LIN {X 0,Y 532.462,Z 881.05,A -85,B 0,C 180,E1 15618.4,E2 15618.4} C_VEL
LIN {X 0,Y 529.556,Z 900.929,A -85,B 0,C 180,E1 15617.745,E2 15617.745} C_VEL
LIN {X 0,Y 525.913,Z 922.421,A -85,B 0,C 180,E1 15616.892,E2 15616.892} C_VEL
LIN {X 0,Y 520.896,Z 948,A -85,B 0,C 180,E1 15615.653,E2 15615.653} C_VEL
LIN {X 0,Y 516.441,Z 968.016,A -85,B 0,C 180,E1 15614.497,E2 15614.497} C_VEL
LIN {X 0,Y 511.868,Z 987.021,A -85,B 0,C 180,E1 15613.228,E2 15613.228} C_VEL
LIN {X 0,Y 506.208,Z 1009.005,A -85,B 0,C 180,E1 15611.528,E2 15611.528} C_VEL
LIN {X 0,Y 500.786,Z 1028.462,A -85,B 0,C 180,E1 15609.762,E2 15609.762} C_VEL
LIN {X 0,Y 495.987,Z 1045.107,A -85,B 0,C 180,E1 15608.041,E2 15608.041} C_VEL
LIN {X 0,Y 490.456,Z 1064.014,A -85,B 0,C 180,E1 15605.81,E2 15605.81} C_VEL
LIN {X 0,Y 489.126,Z 1068.218,A -85,B 0,C 180,E1 15605.252,E2 15605.252} C_VEL
LIN {X 0,Y 486.734,Z 1073.439,A -85,B 0,C 180,E1 15604.629,E2 15604.629} C_VEL
LIN {X 0,Y 477.301,Z 1087.199,A -85,B 0,C 180,E1 15603.072,E2 15603.072} C_VEL
LIN {X 0,Y 475.397,Z 1091.188,A -85,B 0,C 180,E1 15602.478,E2 15602.478} C_VEL
LIN {X 0,Y 471.344,Z 1104.372,A -85,B 0,C 180,E1 15600.183,E2 15600.183} C_VEL
LIN {X 0,Y 467.671,Z 1116.791,A -85,B 0,C 180,E1 15597.731,E2 15597.731} C_VEL
LIN {X 0,Y 463.729,Z 1130.988,A -85,B 0,C 180,E1 15594.456,E2 15594.456} C_VEL
LIN {X 0,Y 461.345,Z 1140.474,A -85,B 0,C 180,E1 15591.887,E2 15591.887} C_VEL
LIN {X 0,Y 459.415,Z 1149.184,A -85,B 0,C 180,E1 15589.164,E2 15589.164} C_VEL
LIN {X 0,Y 457.712,Z 1158.339,A -85,B 0,C 180,E1 15585.717,E2 15585.717} C_VEL
LIN {X 0,Y 456.832,Z 1164.35,A -85,B 0,C 180,E1 15582.9,E2 15582.9} C_VEL
LIN {X 0,Y 456.324,Z 1168.956,A -85,B 0,C 180,E1 15580.223,E2 15580.223} C_VEL
LIN {X 0,Y 456.055,Z 1172.944,A -85,B 0,C 180,E1 15577.179,E2 15577.179} C_VEL
LIN {X 0,Y 455.949,Z 1175.579,A -85,B 0,C 180,E1 15573.898,E2 15573.898} C_VEL
LIN {X 0,Y 455.936,Z 1176.585,A -85,B 0,C 180,E1 15571.257,E2 15571.257} C_VEL
LIN {X 0,Y 455.939,Z 1176.6,A -85,B 0,C 180,E1 15568.744,E2 15568.744} C_VEL
LIN {X 0,Y 455.942,Z 1175.69,A -85,B 0,C 180,E1 15566.225,E2 15566.225} C_VEL
LIN {X 0,Y 456.031,Z 1173.527,A -85,B 0,C 180,E1 15563.327,E2 15563.327} C_VEL
LIN {X 0,Y 456.288,Z 1169.494,A -85,B 0,C 180,E1 15560.031,E2 15560.031} C_VEL
LIN {X 0,Y 456.784,Z 1164.768,A -85,B 0,C 180,E1 15557.228,E2 15557.228} C_VEL
LIN {X 0,Y 457.573,Z 1159.13,A -85,B 0,C 180,E1 15554.539,E2 15554.539} C_VEL
LIN {X 0,Y 459.07,Z 1150.955,A -85,B 0,C 180,E1 15551.327,E2 15551.327} C_VEL
LIN {X 0,Y 461.171,Z 1141.22,A -85,B 0,C 180,E1 15548.238,E2 15548.238} C_VEL
LIN {X 0,Y 463.506,Z 1131.822,A -85,B 0,C 180,E1 15545.668,E2 15545.668} C_VEL
LIN {X 0,Y 467.018,Z 1119.253,A -85,B 0,C 180,E1 15542.688,E2 15542.688} C_VEL
LIN {X 0,Y 471.007,Z 1105.511,A -85,B 0,C 180,E1 15539.935,E2 15539.935} C_VEL
LIN {X 0,Y 474.943,Z 1092.667,A -85,B 0,C 180,E1 15537.674,E2 15537.674} C_VEL
LIN {X 0,Y 480.115,Z 1076.281,A -85,B 0,C 180,E1 15535.14,E2 15535.14} C_VEL
LIN {X 0,Y 485.422,Z 1059.029,A -85,B 0,C 180,E1 15532.86,E2 15532.86} C_VEL
LIN {X 0,Y 490.456,Z 1042.604,A -85,B 0,C 180,E1 15530.954,E2 15530.954} C_VEL
LIN {X 0,Y 496.369,Z 1022.898,A -85,B 0,C 180,E1 15528.953,E2 15528.953} C_VEL
LIN {X 0,Y 502.173,Z 1002.09,A -85,B 0,C 180,E1 15527.16,E2 15527.16} C_VEL
LIN {X 0,Y 506.959,Z 983.945,A -85,B 0,C 180,E1 15525.797,E2 15525.797} C_VEL
LIN {X 0,Y 512.003,Z 963.456,A -85,B 0,C 180,E1 15524.457,E2 15524.457} C_VEL
LIN {X 0,Y 517.286,Z 939.51,A -85,B 0,C 180,E1 15523.141,E2 15523.141} C_VEL
LIN {X 0,Y 521.291,Z 918.889,A -85,B 0,C 180,E1 15522.188,E2 15522.188} C_VEL
LIN {X 0,Y 524.924,Z 897.699,A -85,B 0,C 180,E1 15521.367,E2 15521.367} C_VEL
LIN {X 0,Y 528.667,Z 871.635,A -85,B 0,C 180,E1 15520.555,E2 15520.555} C_VEL
LIN {X 0,Y 531.302,Z 847.596,A -85,B 0,C 180,E1 15519.993,E2 15519.993} C_VEL
LIN {X 0,Y 533.012,Z 825.454,A -85,B 0,C 180,E1 15519.597,E2 15519.597} C_VEL
LIN {X 0,Y 543.801,Z 591.304,A -85,B 0,C 180,E1 15516.126,E2 15516.126} C_VEL
LIN {X 0,Y 549.38,Z 477.095,A -85,B 0,C 180,E1 15514.411,E2 15514.411} C_VEL
LIN {X 0,Y 538.923,Z 460.101,A -85,B 0,C 180,E1 15512.174,E2 15512.174} C_VEL
LIN {X 0,Y 528.718,Z 444.717,A -85,B 0,C 180,E1 15509.77,E2 15509.77} C_VEL
LIN {X 0,Y 520.734,Z 433.186,A -85,B 0,C 180,E1 15507.69,E2 15507.69} C_VEL
LIN {X 0,Y 514.214,Z 424.156,A -85,B 0,C 180,E1 15505.822,E2 15505.822} C_VEL
LIN {X 0,Y 509.213,Z 417.399,A -85,B 0,C 180,E1 15504.26,E2 15504.26} C_VEL
LIN {X 0,Y 503.323,Z 409.516,A -85,B 0,C 180,E1 15502.231,E2 15502.231} C_VEL
LIN {X 0,Y 498.472,Z 403.274,A -85,B 0,C 180,E1 15500.367,E2 15500.367} C_VEL
LIN {X 0,Y 494.802,Z 398.678,A -85,B 0,C 180,E1 15498.803,E2 15498.803} C_VEL
LIN {X 0,Y 490.932,Z 393.536,A -85,B 0,C 180,E1 15496.933,E2 15496.933} C_VEL
LIN {X 0,Y 487.374,Z 389.283,A -85,B 0,C 180,E1 15494.981,E2 15494.981} C_VEL
LIN {X 0,Y 485.876,Z 387.485,A -85,B 0,C 180,E1 15494.054,E2 15494.054} C_VEL
LIN {X 0,Y 481.885,Z 382.272,A -85,B 0,C 180,E1 15491.057,E2 15491.057} C_VEL
LIN {X 0,Y 477.66,Z 376.715,A -85,B 0,C 180,E1 15485.646,E2 15485.646} C_VEL
LIN {X 0,Y 476.978,Z 375.814,A -85,B 0,C 180,E1 15481.081,E2 15481.081} C_VEL
LIN {X 0,Y 478.968,Z 376.994,A -85,B 0,C 180,E1 15476.649,E2 15476.649} C_VEL
LIN {X 0,Y 480.364,Z 378.25,A -85,B 0,C 180,E1 15474.985,E2 15474.985} C_VEL
LIN {X 0,Y 486.543,Z 384.476,A -85,B 0,C 180,E1 15470.119,E2 15470.119} C_VEL
LIN {X 0,Y 490.446,Z 388.953,A -85,B 0,C 180,E1 15467.878,E2 15467.878} C_VEL
LIN {X 0,Y 492.385,Z 390.817,A -85,B 0,C 180,E1 15466.913,E2 15466.913} C_VEL
LIN {X 0,Y 495.897,Z 395.017,A -85,B 0,C 180,E1 15465.282,E2 15465.282} C_VEL
LIN {X 0,Y 497.624,Z 396.68,A -85,B 0,C 180,E1 15464.559,E2 15464.559} C_VEL
LIN {X 0,Y 501.643,Z 401.372,A -85,B 0,C 180,E1 15462.962,E2 15462.962} C_VEL
LIN {X 0,Y 508.034,Z 409.049,A -85,B 0,C 180,E1 15460.692,E2 15460.692} C_VEL
LIN {X 0,Y 512.753,Z 414.817,A -85,B 0,C 180,E1 15459.182,E2 15459.182} C_VEL
LIN {X 0,Y 517.573,Z 420.901,A -85,B 0,C 180,E1 15457.75,E2 15457.75} C_VEL
LIN {X 0,Y 524.781,Z 430.02,A -85,B 0,C 180,E1 15455.787,E2 15455.787} C_VEL
LIN {X 0,Y 534.925,Z 443.868,A -85,B 0,C 180,E1 15453.285,E2 15453.285} C_VEL
LIN {X 0,Y 544.949,Z 458.293,A -85,B 0,C 180,E1 15451.057,E2 15451.057} C_VEL
LIN {X 0,Y 552.935,Z 470.605,A -85,B 0,C 180,E1 15449.413,E2 15449.413} C_VEL
LIN {X 0,Y 541.839,Z 683.901,A -85,B 0,C 180,E1 15446.095,E2 15446.095} C_VEL
LIN {X 0,Y 534.574,Z 826.583,A -85,B 0,C 180,E1 15443.866,E2 15443.866} C_VEL
LIN {X 0,Y 532.122,Z 853.861,A -85,B 0,C 180,E1 15443.33,E2 15443.33} C_VEL
LIN {X 0,Y 528.759,Z 880.247,A -85,B 0,C 180,E1 15442.619,E2 15442.619} C_VEL
LIN {X 0,Y 525.469,Z 902.039,A -85,B 0,C 180,E1 15441.889,E2 15441.889} C_VEL
LIN {X 0,Y 521.778,Z 923.361,A -85,B 0,C 180,E1 15441.035,E2 15441.035} C_VEL
LIN {X 0,Y 516.644,Z 949.664,A -85,B 0,C 180,E1 15439.772,E2 15439.772} C_VEL
LIN {X 0,Y 511.586,Z 972.397,A -85,B 0,C 180,E1 15438.465,E2 15438.465} C_VEL
LIN {X 0,Y 506.827,Z 992.36,A -85,B 0,C 180,E1 15437.143,E2 15437.143} C_VEL
LIN {X 0,Y 501.686,Z 1012.679,A -85,B 0,C 180,E1 15435.608,E2 15435.608} C_VEL
LIN {X 0,Y 495.251,Z 1036.643,A -85,B 0,C 180,E1 15433.507,E2 15433.507} C_VEL
LIN {X 0,Y 490.026,Z 1055.322,A -85,B 0,C 180,E1 15431.618,E2 15431.618} C_VEL
LIN {X 0,Y 485.244,Z 1072.171,A -85,B 0,C 180,E1 15429.7,E2 15429.7} C_VEL
LIN {X 0,Y 479.749,Z 1091.705,A -85,B 0,C 180,E1 15427.186,E2 15427.186} C_VEL
LIN {X 0,Y 474.635,Z 1109.565,A -85,B 0,C 180,E1 15424.519,E2 15424.519} C_VEL
LIN {X 0,Y 470.851,Z 1123.31,A -85,B 0,C 180,E1 15422.209,E2 15422.209} C_VEL
LIN {X 0,Y 467.156,Z 1137.727,A -85,B 0,C 180,E1 15419.49,E2 15419.49} C_VEL
LIN {X 0,Y 463.668,Z 1152.034,A -85,B 0,C 180,E1 15416.374,E2 15416.374} C_VEL
LIN {X 0,Y 461.39,Z 1162.388,A -85,B 0,C 180,E1 15413.771,E2 15413.771} C_VEL
LIN {X 0,Y 459.598,Z 1171.455,A -85,B 0,C 180,E1 15411.17,E2 15411.17} C_VEL
LIN {X 0,Y 458.241,Z 1179.295,A -85,B 0,C 180,E1 15408.576,E2 15408.576} C_VEL
LIN {X 0,Y 457.218,Z 1186.471,A -85,B 0,C 180,E1 15405.795,E2 15405.795} C_VEL
LIN {X 0,Y 456.438,Z 1193.644,A -85,B 0,C 180,E1 15402.396,E2 15402.396} C_VEL
LIN {X 0,Y 456.093,Z 1198.482,A -85,B 0,C 180,E1 15399.336,E2 15399.336} C_VEL
LIN {X 0,Y 455.961,Z 1201.688,A -85,B 0,C 180,E1 15396.585,E2 15396.585} C_VEL
LIN {X 0,Y 455.915,Z 1203.684,A -85,B 0,C 180,E1 15394.024,E2 15394.024} C_VEL
LIN {X 0,Y 455.91,Z 1204.708,A -85,B 0,C 180,E1 15391.508,E2 15391.508} C_VEL
LIN {X 0,Y 455.908,Z 1204.801,A -85,B 0,C 180,E1 15388.994,E2 15388.994} C_VEL
LIN {X 0,Y 455.915,Z 1203.964,A -85,B 0,C 180,E1 15386.479,E2 15386.479} C_VEL
LIN {X 0,Y 455.946,Z 1202.191,A -85,B 0,C 180,E1 15383.957,E2 15383.957} C_VEL
LIN {X 0,Y 456.045,Z 1199.471,A -85,B 0,C 180,E1 15381.426,E2 15381.426} C_VEL
LIN {X 0,Y 456.253,Z 1195.782,A -85,B 0,C 180,E1 15378.88,E2 15378.88} C_VEL
LIN {X 0,Y 456.713,Z 1190.833,A -85,B 0,C 180,E1 15376.194,E2 15376.194} C_VEL
LIN {X 0,Y 457.385,Z 1185.054,A -85,B 0,C 180,E1 15373.62,E2 15373.62} C_VEL
LIN {X 0,Y 458.489,Z 1177.83,A -85,B 0,C 180,E1 15370.906,E2 15370.906} C_VEL
LIN {X 0,Y 460.348,Z 1167.648,A -85,B 0,C 180,E1 15367.66,E2 15367.66} C_VEL
LIN {X 0,Y 462.817,Z 1155.82,A -85,B 0,C 180,E1 15364.537,E2 15364.537} C_VEL
LIN {X 0,Y 465.352,Z 1144.907,A -85,B 0,C 180,E1 15362.02,E2 15362.02} C_VEL
LIN {X 0,Y 468.293,Z 1133.073,A -85,B 0,C 180,E1 15359.6,E2 15359.6} C_VEL
LIN {X 0,Y 472.647,Z 1117.012,A -85,B 0,C 180,E1 15356.682,E2 15356.682} C_VEL
LIN {X 0,Y 477.455,Z 1099.47,A -85,B 0,C 180,E1 15353.937,E2 15353.937} C_VEL
LIN {X 0,Y 481.832,Z 1084.082,A -85,B 0,C 180,E1 15351.801,E2 15351.801} C_VEL
LIN {X 0,Y 486.748,Z 1066.938,A -85,B 0,C 180,E1 15349.679,E2 15349.679} C_VEL
LIN {X 0,Y 493.233,Z 1043.981,A -85,B 0,C 180,E1 15347.211,E2 15347.211} C_VEL
LIN {X 0,Y 498.131,Z 1026.031,A -85,B 0,C 180,E1 15345.53,E2 15345.53} C_VEL
LIN {X 0,Y 502.839,Z 1008.166,A -85,B 0,C 180,E1 15344.042,E2 15344.042} C_VEL
LIN {X 0,Y 507.623,Z 989.113,A -85,B 0,C 180,E1 15342.634,E2 15342.634} C_VEL
LIN {X 0,Y 513.346,Z 964.927,A -85,B 0,C 180,E1 15341.08,E2 15341.08} C_VEL
LIN {X 0,Y 518.424,Z 940.627,A -85,B 0,C 180,E1 15339.773,E2 15339.773} C_VEL
LIN {X 0,Y 522.355,Z 919.986,A -85,B 0,C 180,E1 15338.824,E2 15338.824} C_VEL
LIN {X 0,Y 525.919,Z 899.053,A -85,B 0,C 180,E1 15338.005,E2 15338.005} C_VEL
LIN {X 0,Y 529.858,Z 872.442,A -85,B 0,C 180,E1 15337.15,E2 15337.15} C_VEL
LIN {X 0,Y 532.806,Z 846.446,A -85,B 0,C 180,E1 15336.517,E2 15336.517} C_VEL
LIN {X 0,Y 534.717,Z 823.813,A -85,B 0,C 180,E1 15336.091,E2 15336.091} C_VEL
LIN {X 0,Y 545.542,Z 610.54,A -85,B 0,C 180,E1 15332.769,E2 15332.769} C_VEL
LIN {X 0,Y 552.772,Z 470.258,A -85,B 0,C 180,E1 15330.567,E2 15330.567} C_VEL
LIN {X 0,Y 542.221,Z 454.418,A -85,B 0,C 180,E1 15328.38,E2 15328.38} C_VEL
LIN {X 0,Y 532.873,Z 440.999,A -85,B 0,C 180,E1 15326.255,E2 15326.255} C_VEL
LIN {X 0,Y 523.322,Z 428.23,A -85,B 0,C 180,E1 15323.865,E2 15323.865} C_VEL
LIN {X 0,Y 515.323,Z 417.986,A -85,B 0,C 180,E1 15321.633,E2 15321.633} C_VEL
LIN {X 0,Y 510.35,Z 411.91,A -85,B 0,C 180,E1 15320.111,E2 15320.111} C_VEL
LIN {X 0,Y 506.154,Z 406.806,A -85,B 0,C 180,E1 15318.724,E2 15318.724} C_VEL
LIN {X 0,Y 501.489,Z 401.24,A -85,B 0,C 180,E1 15317.043,E2 15317.043} C_VEL
LIN {X 0,Y 497.404,Z 396.37,A -85,B 0,C 180,E1 15315.418,E2 15315.418} C_VEL
LIN {X 0,Y 492.888,Z 391.636,A -85,B 0,C 180,E1 15313.431,E2 15313.431} C_VEL
LIN {X 0,Y 491.406,Z 389.729,A -85,B 0,C 180,E1 15312.695,E2 15312.695} C_VEL
LIN {X 0,Y 486.891,Z 385.029,A -85,B 0,C 180,E1 15310.232,E2 15310.232} C_VEL
LIN {X 0,Y 485.71,Z 383.571,A -85,B 0,C 180,E1 15309.479,E2 15309.479} C_VEL
LIN {X 0,Y 479.508,Z 377.269,A -85,B 0,C 180,E1 15304.305,E2 15304.305} C_VEL
LIN {X 0,Y 476.828,Z 375.617,A -85,B 0,C 180,E1 15299.519,E2 15299.519} C_VEL
LIN {X 0,Y 477.071,Z 376.199,A -85,B 0,C 180,E1 15295.07,E2 15295.07} C_VEL
LIN {X 0,Y 477.957,Z 377.33,A -85,B 0,C 180,E1 15293.151,E2 15293.151} C_VEL
LIN {X 0,Y 482.557,Z 383.147,A -85,B 0,C 180,E1 15288.102,E2 15288.102} C_VEL
LIN {X 0,Y 487.234,Z 389.112,A -85,B 0,C 180,E1 15284.893,E2 15284.893} C_VEL
LIN {X 0,Y 490.92,Z 393.558,A -85,B 0,C 180,E1 15282.884,E2 15282.884} C_VEL
LIN {X 0,Y 496.633,Z 401.015,A -85,B 0,C 180,E1 15280.23,E2 15280.23} C_VEL
LIN {X 0,Y 500.623,Z 406.102,A -85,B 0,C 180,E1 15278.623,E2 15278.623} C_VEL
LIN {X 0,Y 505.172,Z 411.999,A -85,B 0,C 180,E1 15276.961,E2 15276.961} C_VEL
LIN {X 0,Y 512.277,Z 421.55,A -85,B 0,C 180,E1 15274.632,E2 15274.632} C_VEL
LIN {X 0,Y 518.676,Z 430.345,A -85,B 0,C 180,E1 15272.752,E2 15272.752} C_VEL
LIN {X 0,Y 527.608,Z 443.059,A -85,B 0,C 180,E1 15270.386,E2 15270.386} C_VEL
LIN {X 0,Y 538.197,Z 459.107,A -85,B 0,C 180,E1 15267.872,E2 15267.872} C_VEL
LIN {X 0,Y 548.067,Z 474.977,A -85,B 0,C 180,E1 15265.748,E2 15265.748} C_VEL
LIN {X 0,Y 549.35,Z 477.405,A -85,B 0,C 180,E1 15265.478,E2 15265.478} C_VEL
LIN {X 0,Y 538.35,Z 706.811,A -85,B 0,C 180,E1 15262.067,E2 15262.067} C_VEL
LIN {X 0,Y 532.598,Z 831.176,A -85,B 0,C 180,E1 15260.216,E2 15260.216} C_VEL
LIN {X 0,Y 530.219,Z 858.217,A -85,B 0,C 180,E1 15259.683,E2 15259.683} C_VEL
LIN {X 0,Y 527.373,Z 880.936,A -85,B 0,C 180,E1 15259.078,E2 15259.078} C_VEL
LIN {X 0,Y 524.411,Z 900.63,A -85,B 0,C 180,E1 15258.43,E2 15258.43} C_VEL
LIN {X 0,Y 520.708,Z 921.873,A -85,B 0,C 180,E1 15257.589,E2 15257.589} C_VEL
LIN {X 0,Y 515.429,Z 948.057,A -85,B 0,C 180,E1 15256.321,E2 15256.321} C_VEL
LIN {X 0,Y 510.955,Z 967.573,A -85,B 0,C 180,E1 15255.192,E2 15255.192} C_VEL
LIN {X 0,Y 506.155,Z 986.915,A -85,B 0,C 180,E1 15253.898,E2 15253.898} C_VEL
LIN {X 0,Y 500.279,Z 1008.979,A -85,B 0,C 180,E1 15252.187,E2 15252.187} C_VEL
LIN {X 0,Y 494.655,Z 1028.456,A -85,B 0,C 180,E1 15250.408,E2 15250.408} C_VEL
LIN {X 0,Y 489.663,Z 1045.152,A -85,B 0,C 180,E1 15248.671,E2 15248.671} C_VEL
LIN {X 0,Y 483.962,Z 1063.92,A -85,B 0,C 180,E1 15246.44,E2 15246.44} C_VEL
LIN {X 0,Y 478.537,Z 1081.053,A -85,B 0,C 180,E1 15244.054,E2 15244.054} C_VEL
LIN {X 0,Y 475.397,Z 1091.188,A -85,B 0,C 180,E1 15242.478,E2 15242.478} C_VEL
LIN {X 0,Y 473.094,Z 1095.843,A -85,B 0,C 180,E1 15241.776,E2 15241.776} C_VEL
LIN {X 0,Y 463.841,Z 1108.186,A -85,B 0,C 180,E1 15239.993,E2 15239.993} C_VEL
LIN {X 0,Y 462.049,Z 1111.733,A -85,B 0,C 180,E1 15239.332,E2 15239.332} C_VEL
LIN {X 0,Y 458.366,Z 1123.819,A -85,B 0,C 180,E1 15236.703,E2 15236.703} C_VEL
LIN {X 0,Y 455.419,Z 1134.273,A -85,B 0,C 180,E1 15234.102,E2 15234.102} C_VEL
LIN {X 0,Y 452.577,Z 1145.51,A -85,B 0,C 180,E1 15230.836,E2 15230.836} C_VEL
LIN {X 0,Y 450.692,Z 1154.074,A -85,B 0,C 180,E1 15227.828,E2 15227.828} C_VEL
LIN {X 0,Y 449.497,Z 1160.654,A -85,B 0,C 180,E1 15225.086,E2 15225.086} C_VEL
LIN {X 0,Y 448.613,Z 1167.046,A -85,B 0,C 180,E1 15221.833,E2 15221.833} C_VEL
LIN {X 0,Y 448.177,Z 1171.674,A -85,B 0,C 180,E1 15218.597,E2 15218.597} C_VEL
LIN {X 0,Y 447.993,Z 1174.46,A -85,B 0,C 180,E1 15215.893,E2 15215.893} C_VEL
LIN {X 0,Y 447.945,Z 1176.219,A -85,B 0,C 180,E1 15213.199,E2 15213.199} C_VEL
LIN {X 0,Y 447.936,Z 1177.029,A -85,B 0,C 180,E1 15210.128,E2 15210.128} C_VEL
LIN {X 0,Y 447.943,Z 1176.331,A -85,B 0,C 180,E1 15206.929,E2 15206.929} C_VEL
LIN {X 0,Y 447.993,Z 1174.539,A -85,B 0,C 180,E1 15204.107,E2 15204.107} C_VEL
LIN {X 0,Y 448.169,Z 1171.783,A -85,B 0,C 180,E1 15201.404,E2 15201.404} C_VEL
LIN {X 0,Y 448.547,Z 1167.582,A -85,B 0,C 180,E1 15198.427,E2 15198.427} C_VEL
LIN {X 0,Y 449.424,Z 1161.15,A -85,B 0,C 180,E1 15195.044,E2 15195.044} C_VEL
LIN {X 0,Y 450.582,Z 1154.652,A -85,B 0,C 180,E1 15192.301,E2 15192.301} C_VEL
LIN {X 0,Y 452.224,Z 1146.949,A -85,B 0,C 180,E1 15189.553,E2 15189.553} C_VEL
LIN {X 0,Y 454.955,Z 1136.099,A -85,B 0,C 180,E1 15186.285,E2 15186.285} C_VEL
LIN {X 0,Y 458.093,Z 1124.745,A -85,B 0,C 180,E1 15183.42,E2 15183.42} C_VEL
LIN {X 0,Y 461.456,Z 1113.604,A -85,B 0,C 180,E1 15180.964,E2 15180.964} C_VEL
LIN {X 0,Y 466.102,Z 1098.989,A -85,B 0,C 180,E1 15178.149,E2 15178.149} C_VEL
LIN {X 0,Y 471.039,Z 1083.585,A -85,B 0,C 180,E1 15175.623,E2 15175.623} C_VEL
LIN {X 0,Y 475.822,Z 1068.929,A -85,B 0,C 180,E1 15173.51,E2 15173.51} C_VEL
LIN {X 0,Y 481.805,Z 1050.577,A -85,B 0,C 180,E1 15171.191,E2 15171.191} C_VEL
LIN {X 0,Y 487.874,Z 1030.932,A -85,B 0,C 180,E1 15169.081,E2 15169.081} C_VEL
LIN {X 0,Y 492.905,Z 1014.172,A -85,B 0,C 180,E1 15167.507,E2 15167.507} C_VEL
LIN {X 0,Y 498.692,Z 993.945,A -85,B 0,C 180,E1 15165.843,E2 15165.843} C_VEL
LIN {X 0,Y 504.647,Z 970.976,A -85,B 0,C 180,E1 15164.246,E2 15164.246} C_VEL
LIN {X 0,Y 509.316,Z 951.469,A -85,B 0,C 180,E1 15163.089,E2 15163.089} C_VEL
LIN {X 0,Y 513.751,Z 931.077,A -85,B 0,C 180,E1 15162.048,E2 15162.048} C_VEL
LIN {X 0,Y 518.582,Z 905.394,A -85,B 0,C 180,E1 15160.963,E2 15160.963} C_VEL
LIN {X 0,Y 521.939,Z 884.167,A -85,B 0,C 180,E1 15160.238,E2 15160.238} C_VEL
LIN {X 0,Y 524.617,Z 863.87,A -85,B 0,C 180,E1 15159.672,E2 15159.672} C_VEL
LIN {X 0,Y 527.172,Z 839.566,A -85,B 0,C 180,E1 15159.145,E2 15159.145} C_VEL
LIN {X 0,Y 529.271,Z 803.306,A -85,B 0,C 180,E1 15158.57,E2 15158.57} C_VEL
LIN {X 0,Y 540.117,Z 575.69,A -85,B 0,C 180,E1 15155.184,E2 15155.184} C_VEL
LIN {X 0,Y 544.866,Z 481.213,A -85,B 0,C 180,E1 15153.751,E2 15153.751} C_VEL
LIN {X 0,Y 535.364,Z 465.745,A -85,B 0,C 180,E1 15151.656,E2 15151.656} C_VEL
LIN {X 0,Y 525.934,Z 451.284,A -85,B 0,C 180,E1 15149.374,E2 15149.374} C_VEL
LIN {X 0,Y 518.091,Z 439.848,A -85,B 0,C 180,E1 15147.282,E2 15147.282} C_VEL
LIN {X 0,Y 512.035,Z 431.315,A -85,B 0,C 180,E1 15145.505,E2 15145.505} C_VEL
LIN {X 0,Y 505.61,Z 422.408,A -85,B 0,C 180,E1 15143.422,E2 15143.422} C_VEL
LIN {X 0,Y 501.184,Z 416.583,A -85,B 0,C 180,E1 15141.844,E2 15141.844} C_VEL
LIN {X 0,Y 496.7,Z 410.664,A -85,B 0,C 180,E1 15140.074,E2 15140.074} C_VEL
LIN {X 0,Y 493.095,Z 406.104,A -85,B 0,C 180,E1 15138.503,E2 15138.503} C_VEL
LIN {X 0,Y 489.413,Z 401.142,A -85,B 0,C 180,E1 15136.681,E2 15136.681} C_VEL
LIN {X 0,Y 485.846,Z 396.679,A -85,B 0,C 180,E1 15134.663,E2 15134.663} C_VEL
LIN {X 0,Y 480.729,Z 390.107,A -85,B 0,C 180,E1 15130.911,E2 15130.911} C_VEL
LIN {X 0,Y 476.638,Z 384.614,A -85,B 0,C 180,E1 15125.538,E2 15125.538} C_VEL
LIN {X 0,Y 476.019,Z 383.758,A -85,B 0,C 180,E1 15120.963,E2 15120.963} C_VEL
LIN {X 0,Y 478.172,Z 385.043,A -85,B 0,C 180,E1 15116.403,E2 15116.403} C_VEL
LIN {X 0,Y 479.485,Z 386.415,A -85,B 0,C 180,E1 15114.855,E2 15114.855} C_VEL
LIN {X 0,Y 485.192,Z 392.155,A -85,B 0,C 180,E1 15110.331,E2 15110.331} C_VEL
LIN {X 0,Y 489.244,Z 396.837,A -85,B 0,C 180,E1 15107.968,E2 15107.968} C_VEL
LIN {X 0,Y 490.93,Z 398.526,A -85,B 0,C 180,E1 15107.113,E2 15107.113} C_VEL
LIN {X 0,Y 494.526,Z 402.811,A -85,B 0,C 180,E1 15105.42,E2 15105.42} C_VEL
LIN {X 0,Y 496.223,Z 404.609,A -85,B 0,C 180,E1 15104.694,E2 15104.694} C_VEL
LIN {X 0,Y 501.221,Z 410.498,A -85,B 0,C 180,E1 15102.708,E2 15102.708} C_VEL
LIN {X 0,Y 506.311,Z 416.724,A -85,B 0,C 180,E1 15100.893,E2 15100.893} C_VEL
LIN {X 0,Y 510.814,Z 422.288,A -85,B 0,C 180,E1 15099.429,E2 15099.429} C_VEL
LIN {X 0,Y 515.576,Z 428.38,A -85,B 0,C 180,E1 15097.989,E2 15097.989} C_VEL
LIN {X 0,Y 522.515,Z 437.285,A -85,B 0,C 180,E1 15096.066,E2 15096.066} C_VEL
LIN {X 0,Y 532.238,Z 450.725,A -85,B 0,C 180,E1 15093.621,E2 15093.621} C_VEL
LIN {X 0,Y 542.138,Z 465.167,A -85,B 0,C 180,E1 15091.375,E2 15091.375} C_VEL
LIN {X 0,Y 548.391,Z 474.999,A -85,B 0,C 180,E1 15090.051,E2 15090.051} C_VEL
LIN {X 0,Y 536.927,Z 688.4,A -85,B 0,C 180,E1 15086.718,E2 15086.718} C_VEL
LIN {X 0,Y 529.646,Z 826.679,A -85,B 0,C 180,E1 15084.547,E2 15084.547} C_VEL
LIN {X 0,Y 527.109,Z 854.091,A -85,B 0,C 180,E1 15084.007,E2 15084.007} C_VEL
LIN {X 0,Y 523.677,Z 880.287,A -85,B 0,C 180,E1 15083.299,E2 15083.299} C_VEL
LIN {X 0,Y 520.312,Z 901.929,A -85,B 0,C 180,E1 15082.573,E2 15082.573} C_VEL
LIN {X 0,Y 516.536,Z 923.116,A -85,B 0,C 180,E1 15081.724,E2 15081.724} C_VEL
LIN {X 0,Y 511.332,Z 949.047,A -85,B 0,C 180,E1 15080.481,E2 15080.481} C_VEL
LIN {X 0,Y 505.911,Z 972.651,A -85,B 0,C 180,E1 15079.118,E2 15079.118} C_VEL
LIN {X 0,Y 501.16,Z 991.953,A -85,B 0,C 180,E1 15077.832,E2 15077.832} C_VEL
LIN {X 0,Y 496.053,Z 1011.473,A -85,B 0,C 180,E1 15076.354,E2 15076.354} C_VEL
LIN {X 0,Y 489.551,Z 1034.938,A -85,B 0,C 180,E1 15074.307,E2 15074.307} C_VEL
LIN {X 0,Y 483.912,Z 1054.308,A -85,B 0,C 180,E1 15072.345,E2 15072.345} C_VEL
LIN {X 0,Y 478.907,Z 1071.214,A -85,B 0,C 180,E1 15070.411,E2 15070.411} C_VEL
LIN {X 0,Y 473.735,Z 1088.691,A -85,B 0,C 180,E1 15068.159,E2 15068.159} C_VEL
LIN {X 0,Y 468.048,Z 1107.914,A -85,B 0,C 180,E1 15065.307,E2 15065.307} C_VEL
LIN {X 0,Y 463.915,Z 1122.151,A -85,B 0,C 180,E1 15062.897,E2 15062.897} C_VEL
LIN {X 0,Y 460.461,Z 1134.589,A -85,B 0,C 180,E1 15060.539,E2 15060.539} C_VEL
LIN {X 0,Y 456.978,Z 1148.192,A -85,B 0,C 180,E1 15057.636,E2 15057.636} C_VEL
LIN {X 0,Y 453.828,Z 1161.463,A -85,B 0,C 180,E1 15054.33,E2 15054.33} C_VEL
LIN {X 0,Y 451.904,Z 1170.658,A -85,B 0,C 180,E1 15051.673,E2 15051.673} C_VEL
LIN {X 0,Y 450.46,Z 1178.567,A -85,B 0,C 180,E1 15049.044,E2 15049.044} C_VEL
LIN {X 0,Y 449.393,Z 1185.361,A -85,B 0,C 180,E1 15046.413,E2 15046.413} C_VEL
LIN {X 0,Y 448.68,Z 1191.316,A -85,B 0,C 180,E1 15043.663,E2 15043.663} C_VEL
LIN {X 0,Y 448.187,Z 1196.991,A -85,B 0,C 180,E1 15040.411,E2 15040.411} C_VEL
LIN {X 0,Y 447.974,Z 1201.111,A -85,B 0,C 180,E1 15037.051,E2 15037.051} C_VEL
LIN {X 0,Y 447.92,Z 1203.361,A -85,B 0,C 180,E1 15034.224,E2 15034.224} C_VEL
LIN {X 0,Y 447.911,Z 1204.436,A -85,B 0,C 180,E1 15031.663,E2 15031.663} C_VEL
LIN {X 0,Y 447.908,Z 1204.577,A -85,B 0,C 180,E1 15029.104,E2 15029.104} C_VEL
LIN {X 0,Y 447.917,Z 1203.714,A -85,B 0,C 180,E1 15026.416,E2 15026.416} C_VEL
LIN {X 0,Y 447.951,Z 1201.935,A -85,B 0,C 180,E1 15023.849,E2 15023.849} C_VEL
LIN {X 0,Y 448.054,Z 1199.204,A -85,B 0,C 180,E1 15021.271,E2 15021.271} C_VEL
LIN {X 0,Y 448.275,Z 1195.5,A -85,B 0,C 180,E1 15018.68,E2 15018.68} C_VEL
LIN {X 0,Y 448.736,Z 1190.793,A -85,B 0,C 180,E1 15016.075,E2 15016.075} C_VEL
LIN {X 0,Y 449.436,Z 1185.044,A -85,B 0,C 180,E1 15013.455,E2 15013.455} C_VEL
LIN {X 0,Y 450.589,Z 1177.838,A -85,B 0,C 180,E1 15010.692,E2 15010.692} C_VEL
LIN {X 0,Y 452.466,Z 1167.953,A -85,B 0,C 180,E1 15007.478,E2 15007.478} C_VEL
LIN {X 0,Y 455.107,Z 1155.88,A -85,B 0,C 180,E1 15004.214,E2 15004.214} C_VEL
LIN {X 0,Y 457.835,Z 1144.603,A -85,B 0,C 180,E1 15001.569,E2 15001.569} C_VEL
LIN {X 0,Y 461.011,Z 1132.611,A -85,B 0,C 180,E1 14999.067,E2 14999.067} C_VEL
LIN {X 0,Y 465.426,Z 1117.066,A -85,B 0,C 180,E1 14996.192,E2 14996.192} C_VEL
LIN {X 0,Y 470.343,Z 1099.999,A -85,B 0,C 180,E1 14993.47,E2 14993.47} C_VEL
LIN {X 0,Y 474.917,Z 1084.606,A -85,B 0,C 180,E1 14991.296,E2 14991.296} C_VEL
LIN {X 0,Y 479.692,Z 1068.587,A -85,B 0,C 180,E1 14989.275,E2 14989.275} C_VEL
LIN {X 0,Y 485.84,Z 1047.993,A -85,B 0,C 180,E1 14986.981,E2 14986.981} C_VEL
LIN {X 0,Y 491.792,Z 1026.909,A -85,B 0,C 180,E1 14984.965,E2 14984.965} C_VEL
LIN {X 0,Y 496.619,Z 1009.281,A -85,B 0,C 180,E1 14983.477,E2 14983.477} C_VEL
LIN {X 0,Y 501.369,Z 991.052,A -85,B 0,C 180,E1 14982.108,E2 14982.108} C_VEL
LIN {X 0,Y 506.393,Z 970.579,A -85,B 0,C 180,E1 14980.756,E2 14980.756} C_VEL
LIN {X 0,Y 512.247,Z 944.525,A -85,B 0,C 180,E1 14979.29,E2 14979.29} C_VEL
LIN {X 0,Y 516.742,Z 921.818,A -85,B 0,C 180,E1 14978.224,E2 14978.224} C_VEL
LIN {X 0,Y 520.426,Z 901.019,A -85,B 0,C 180,E1 14977.397,E2 14977.397} C_VEL
LIN {X 0,Y 523.856,Z 878.838,A -85,B 0,C 180,E1 14976.66,E2 14976.66} C_VEL
LIN {X 0,Y 527.386,Z 850.986,A -85,B 0,C 180,E1 14975.93,E2 14975.93} C_VEL
LIN {X 0,Y 529.658,Z 825.826,A -85,B 0,C 180,E1 14975.442,E2 14975.442} C_VEL
LIN {X 0,Y 540.247,Z 624.464,A -85,B 0,C 180,E1 14972.288,E2 14972.288} C_VEL
LIN {X 0,Y 548.34,Z 474.693,A -85,B 0,C 180,E1 14969.949,E2 14969.949} C_VEL
LIN {X 0,Y 536.551,Z 456.942,A -85,B 0,C 180,E1 14967.406,E2 14967.406} C_VEL
LIN {X 0,Y 527.28,Z 443.875,A -85,B 0,C 180,E1 14965.197,E2 14965.197} C_VEL
LIN {X 0,Y 518.102,Z 431.461,A -85,B 0,C 180,E1 14962.765,E2 14962.765} C_VEL
LIN {X 0,Y 509.027,Z 419.974,A -85,B 0,C 180,E1 14960.046,E2 14960.046} C_VEL
LIN {X 0,Y 504.065,Z 414.015,A -85,B 0,C 180,E1 14958.385,E2 14958.385} C_VEL
LIN {X 0,Y 499.625,Z 408.646,A -85,B 0,C 180,E1 14956.749,E2 14956.749} C_VEL
LIN {X 0,Y 494.884,Z 403.11,A -85,B 0,C 180,E1 14954.808,E2 14954.808} C_VEL
LIN {X 0,Y 491.086,Z 398.824,A -85,B 0,C 180,E1 14953.062,E2 14953.062} C_VEL
LIN {X 0,Y 489.964,Z 397.43,A -85,B 0,C 180,E1 14952.493,E2 14952.493} C_VEL
LIN {X 0,Y 485.526,Z 392.707,A -85,B 0,C 180,E1 14950.022,E2 14950.022} C_VEL
LIN {X 0,Y 484.363,Z 391.323,A -85,B 0,C 180,E1 14949.266,E2 14949.266} C_VEL
LIN {X 0,Y 478.422,Z 385.155,A -85,B 0,C 180,E1 14944.195,E2 14944.195} C_VEL
LIN {X 0,Y 475.821,Z 383.549,A -85,B 0,C 180,E1 14939.398,E2 14939.398} C_VEL
LIN {X 0,Y 476.141,Z 384.191,A -85,B 0,C 180,E1 14934.94,E2 14934.94} C_VEL
LIN {X 0,Y 476.979,Z 385.348,A -85,B 0,C 180,E1 14933.137,E2 14933.137} C_VEL
LIN {X 0,Y 481.374,Z 390.961,A -85,B 0,C 180,E1 14928.255,E2 14928.255} C_VEL
LIN {X 0,Y 485.883,Z 396.823,A -85,B 0,C 180,E1 14925.094,E2 14925.094} C_VEL
LIN {X 0,Y 489.628,Z 401.368,A -85,B 0,C 180,E1 14923.021,E2 14923.021} C_VEL
LIN {X 0,Y 495.405,Z 409.108,A -85,B 0,C 180,E1 14920.302,E2 14920.302} C_VEL
LIN {X 0,Y 498.948,Z 413.692,A -85,B 0,C 180,E1 14918.855,E2 14918.855} C_VEL
LIN {X 0,Y 503.37,Z 419.507,A -85,B 0,C 180,E1 14917.21,E2 14917.21} C_VEL
LIN {X 0,Y 510.206,Z 428.834,A -85,B 0,C 180,E1 14914.925,E2 14914.925} C_VEL
LIN {X 0,Y 516.431,Z 437.517,A -85,B 0,C 180,E1 14913.06,E2 14913.06} C_VEL
LIN {X 0,Y 525.324,Z 450.408,A -85,B 0,C 180,E1 14910.658,E2 14910.658} C_VEL
LIN {X 0,Y 535.611,Z 466.172,A -85,B 0,C 180,E1 14908.171,E2 14908.171} C_VEL
LIN {X 0,Y 544.889,Z 481.344,A -85,B 0,C 180,E1 14906.132,E2 14906.132} C_VEL
LIN {X 0,Y 533.478,Z 711.175,A -85,B 0,C 180,E1 14902.701,E2 14902.701} C_VEL
LIN {X 0,Y 527.72,Z 831.166,A -85,B 0,C 180,E1 14900.904,E2 14900.904} C_VEL
LIN {X 0,Y 525.272,Z 858.21,A -85,B 0,C 180,E1 14900.371,E2 14900.371} C_VEL
LIN {X 0,Y 522.344,Z 880.922,A -85,B 0,C 180,E1 14899.766,E2 14899.766} C_VEL
LIN {X 0,Y 519.196,Z 901.222,A -85,B 0,C 180,E1 14899.096,E2 14899.096} C_VEL
LIN {X 0,Y 515.354,Z 922.588,A -85,B 0,C 180,E1 14898.245,E2 14898.245} C_VEL
LIN {X 0,Y 509.999,Z 948.263,A -85,B 0,C 180,E1 14896.994,E2 14896.994} C_VEL
LIN {X 0,Y 505.224,Z 968.436,A -85,B 0,C 180,E1 14895.819,E2 14895.819} C_VEL
LIN {X 0,Y 500.246,Z 987.835,A -85,B 0,C 180,E1 14894.51,E2 14894.51} C_VEL
LIN {X 0,Y 493.712,Z 1011.303,A -85,B 0,C 180,E1 14892.652,E2 14892.652} C_VEL
LIN {X 0,Y 488.217,Z 1029.68,A -85,B 0,C 180,E1 14890.948,E2 14890.948} C_VEL
LIN {X 0,Y 482.862,Z 1046.951,A -85,B 0,C 180,E1 14889.12,E2 14889.12} C_VEL
LIN {X 0,Y 476.608,Z 1066.534,A -85,B 0,C 180,E1 14886.72,E2 14886.72} C_VEL
LIN {X 0,Y 471.738,Z 1081.397,A -85,B 0,C 180,E1 14884.614,E2 14884.614} C_VEL
LIN {X 0,Y 467.164,Z 1095.495,A -85,B 0,C 180,E1 14882.349,E2 14882.349} C_VEL
LIN {X 0,Y 462.375,Z 1110.731,A -85,B 0,C 180,E1 14879.541,E2 14879.541} C_VEL
LIN {X 0,Y 462.049,Z 1111.733,A -85,B 0,C 180,E1 14879.332,E2 14879.332} C_VEL
LIN {X 0,Y 459.887,Z 1115.797,A -85,B 0,C 180,E1 14878.553,E2 14878.553} C_VEL
LIN {X 0,Y 450.982,Z 1126.66,A -85,B 0,C 180,E1 14876.548,E2 14876.548} C_VEL
LIN {X 0,Y 449.349,Z 1129.716,A -85,B 0,C 180,E1 14875.824,E2 14875.824} C_VEL
LIN {X 0,Y 446.217,Z 1140.62,A -85,B 0,C 180,E1 14872.809,E2 14872.809} C_VEL
LIN {X 0,Y 444.029,Z 1149.305,A -85,B 0,C 180,E1 14870.016,E2 14870.016} C_VEL
LIN {X 0,Y 442.119,Z 1158.309,A -85,B 0,C 180,E1 14866.556,E2 14866.556} C_VEL
LIN {X 0,Y 441.01,Z 1164.787,A -85,B 0,C 180,E1 14863.427,E2 14863.427} C_VEL
LIN {X 0,Y 440.408,Z 1169.483,A -85,B 0,C 180,E1 14860.597,E2 14860.597} C_VEL
LIN {X 0,Y 440.097,Z 1173.459,A -85,B 0,C 180,E1 14857.441,E2 14857.441} C_VEL
LIN {X 0,Y 439.961,Z 1176.078,A -85,B 0,C 180,E1 14854.04,E2 14854.04} C_VEL
LIN {X 0,Y 439.942,Z 1177.079,A -85,B 0,C 180,E1 14851.303,E2 14851.303} C_VEL
LIN {X 0,Y 439.946,Z 1177.095,A -85,B 0,C 180,E1 14848.698,E2 14848.698} C_VEL
LIN {X 0,Y 439.954,Z 1176.19,A -85,B 0,C 180,E1 14846.091,E2 14846.091} C_VEL
LIN {X 0,Y 440.048,Z 1174.131,A -85,B 0,C 180,E1 14843.203,E2 14843.203} C_VEL
LIN {X 0,Y 440.342,Z 1170.215,A -85,B 0,C 180,E1 14839.799,E2 14839.799} C_VEL
LIN {X 0,Y 440.938,Z 1165.302,A -85,B 0,C 180,E1 14836.76,E2 14836.76} C_VEL
LIN {X 0,Y 441.855,Z 1159.676,A -85,B 0,C 180,E1 14833.974,E2 14833.974} C_VEL
LIN {X 0,Y 443.552,Z 1151.522,A -85,B 0,C 180,E1 14830.648,E2 14830.648} C_VEL
LIN {X 0,Y 445.906,Z 1141.802,A -85,B 0,C 180,E1 14827.453,E2 14827.453} C_VEL
LIN {X 0,Y 448.512,Z 1132.415,A -85,B 0,C 180,E1 14824.799,E2 14824.799} C_VEL
LIN {X 0,Y 452.325,Z 1120.05,A -85,B 0,C 180,E1 14821.768,E2 14821.768} C_VEL
LIN {X 0,Y 456.888,Z 1105.835,A -85,B 0,C 180,E1 14818.837,E2 14818.837} C_VEL
LIN {X 0,Y 461.334,Z 1092.569,A -85,B 0,C 180,E1 14816.45,E2 14816.45} C_VEL
LIN {X 0,Y 467.128,Z 1075.596,A -85,B 0,C 180,E1 14813.789,E2 14813.789} C_VEL
LIN {X 0,Y 472.952,Z 1058.207,A -85,B 0,C 180,E1 14811.466,E2 14811.466} C_VEL
LIN {X 0,Y 478.217,Z 1042.265,A -85,B 0,C 180,E1 14809.597,E2 14809.597} C_VEL
LIN {X 0,Y 484.785,Z 1021.789,A -85,B 0,C 180,E1 14807.509,E2 14807.509} C_VEL
LIN {X 0,Y 490.609,Z 1002.247,A -85,B 0,C 180,E1 14805.813,E2 14805.813} C_VEL
LIN {X 0,Y 495.498,Z 984.886,A -85,B 0,C 180,E1 14804.493,E2 14804.493} C_VEL
LIN {X 0,Y 500.621,Z 965.359,A -85,B 0,C 180,E1 14803.197,E2 14803.197} C_VEL
LIN {X 0,Y 506.703,Z 939.626,A -85,B 0,C 180,E1 14801.763,E2 14801.763} C_VEL
LIN {X 0,Y 511.049,Z 918.479,A -85,B 0,C 180,E1 14800.785,E2 14800.785} C_VEL
LIN {X 0,Y 514.897,Z 897.154,A -85,B 0,C 180,E1 14799.958,E2 14799.958} C_VEL
LIN {X 0,Y 519.039,Z 869.339,A -85,B 0,C 180,E1 14799.107,E2 14799.107} C_VEL
LIN {X 0,Y 521.638,Z 846.653,A -85,B 0,C 180,E1 14798.584,E2 14798.584} C_VEL
LIN {X 0,Y 523.468,Z 823.805,A -85,B 0,C 180,E1 14798.178,E2 14798.178} C_VEL
LIN {X 0,Y 535.074,Z 589.3,A -85,B 0,C 180,E1 14794.67,E2 14794.67} C_VEL
LIN {X 0,Y 540.486,Z 485.434,A -85,B 0,C 180,E1 14793.093,E2 14793.093} C_VEL
LIN {X 0,Y 529.694,Z 467.828,A -85,B 0,C 180,E1 14790.611,E2 14790.611} C_VEL
LIN {X 0,Y 519.738,Z 452.688,A -85,B 0,C 180,E1 14788.059,E2 14788.059} C_VEL
LIN {X 0,Y 510.737,Z 439.567,A -85,B 0,C 180,E1 14785.45,E2 14785.45} C_VEL
LIN {X 0,Y 503.55,Z 429.596,A -85,B 0,C 180,E1 14783.09,E2 14783.09} C_VEL
LIN {X 0,Y 499.348,Z 423.967,A -85,B 0,C 180,E1 14781.558,E2 14781.558} C_VEL
LIN {X 0,Y 494.939,Z 418.059,A -85,B 0,C 180,E1 14779.779,E2 14779.779} C_VEL
LIN {X 0,Y 491.402,Z 413.525,A -85,B 0,C 180,E1 14778.2,E2 14778.2} C_VEL
LIN {X 0,Y 488.061,Z 408.89,A -85,B 0,C 180,E1 14776.509,E2 14776.509} C_VEL
LIN {X 0,Y 484.507,Z 404.392,A -85,B 0,C 180,E1 14774.46,E2 14774.46} C_VEL
LIN {X 0,Y 479.631,Z 397.991,A -85,B 0,C 180,E1 14770.814,E2 14770.814} C_VEL
LIN {X 0,Y 475.619,Z 392.515,A -85,B 0,C 180,E1 14765.429,E2 14765.429} C_VEL
LIN {X 0,Y 475.063,Z 391.702,A -85,B 0,C 180,E1 14760.844,E2 14760.844} C_VEL
LIN {X 0,Y 477.288,Z 393.05,A -85,B 0,C 180,E1 14756.276,E2 14756.276} C_VEL
LIN {X 0,Y 478.828,Z 394.928,A -85,B 0,C 180,E1 14754.488,E2 14754.488} C_VEL
LIN {X 0,Y 483.934,Z 399.972,A -85,B 0,C 180,E1 14750.486,E2 14750.486} C_VEL
LIN {X 0,Y 488.044,Z 404.72,A -85,B 0,C 180,E1 14748.058,E2 14748.058} C_VEL
LIN {X 0,Y 489.484,Z 406.232,A -85,B 0,C 180,E1 14747.315,E2 14747.315} C_VEL
LIN {X 0,Y 493.288,Z 410.717,A -85,B 0,C 180,E1 14745.503,E2 14745.503} C_VEL
LIN {X 0,Y 494.827,Z 412.52,A -85,B 0,C 180,E1 14744.83,E2 14744.83} C_VEL
LIN {X 0,Y 499.566,Z 418.149,A -85,B 0,C 180,E1 14742.919,E2 14742.919} C_VEL
LIN {X 0,Y 504.442,Z 424.177,A -85,B 0,C 180,E1 14741.15,E2 14741.15} C_VEL
LIN {X 0,Y 508.968,Z 429.869,A -85,B 0,C 180,E1 14739.652,E2 14739.652} C_VEL
LIN {X 0,Y 513.765,Z 436.089,A -85,B 0,C 180,E1 14738.178,E2 14738.178} C_VEL
LIN {X 0,Y 520.638,Z 445.086,A -85,B 0,C 180,E1 14736.245,E2 14736.245} C_VEL
LIN {X 0,Y 529.668,Z 457.735,A -85,B 0,C 180,E1 14733.936,E2 14733.936} C_VEL
LIN {X 0,Y 539.345,Z 472.039,A -85,B 0,C 180,E1 14731.697,E2 14731.697} C_VEL
LIN {X 0,Y 543.914,Z 479.375,A -85,B 0,C 180,E1 14730.7,E2 14730.7} C_VEL
LIN {X 0,Y 532.127,Z 692.058,A -85,B 0,C 180,E1 14727.366,E2 14727.366} C_VEL
LIN {X 0,Y 524.802,Z 826.684,A -85,B 0,C 180,E1 14725.243,E2 14725.243} C_VEL
LIN {X 0,Y 522.202,Z 854.102,A -85,B 0,C 180,E1 14724.701,E2 14724.701} C_VEL
LIN {X 0,Y 518.693,Z 880.192,A -85,B 0,C 180,E1 14723.997,E2 14723.997} C_VEL
LIN {X 0,Y 515.232,Z 901.833,A -85,B 0,C 180,E1 14723.271,E2 14723.271} C_VEL
LIN {X 0,Y 511.447,Z 922.51,A -85,B 0,C 180,E1 14722.443,E2 14722.443} C_VEL
LIN {X 0,Y 506.252,Z 947.838,A -85,B 0,C 180,E1 14721.237,E2 14721.237} C_VEL
LIN {X 0,Y 500.567,Z 971.876,A -85,B 0,C 180,E1 14719.851,E2 14719.851} C_VEL
LIN {X 0,Y 495.607,Z 991.43,A -85,B 0,C 180,E1 14718.546,E2 14718.546} C_VEL
LIN {X 0,Y 490.735,Z 1009.478,A -85,B 0,C 180,E1 14717.181,E2 14717.181} C_VEL
LIN {X 0,Y 485.229,Z 1028.858,A -85,B 0,C 180,E1 14715.523,E2 14715.523} C_VEL
LIN {X 0,Y 478.26,Z 1052.157,A -85,B 0,C 180,E1 14713.213,E2 14713.213} C_VEL
LIN {X 0,Y 472.995,Z 1069.234,A -85,B 0,C 180,E1 14711.265,E2 14711.265} C_VEL
LIN {X 0,Y 468.042,Z 1085.167,A -85,B 0,C 180,E1 14709.223,E2 14709.223} C_VEL
LIN {X 0,Y 462.644,Z 1102.669,A -85,B 0,C 180,E1 14706.695,E2 14706.695} C_VEL
LIN {X 0,Y 457.279,Z 1120.31,A -85,B 0,C 180,E1 14703.737,E2 14703.737} C_VEL
LIN {X 0,Y 453.387,Z 1133.531,A -85,B 0,C 180,E1 14701.215,E2 14701.215} C_VEL
LIN {X 0,Y 450.08,Z 1145.46,A -85,B 0,C 180,E1 14698.654,E2 14698.654} C_VEL
LIN {X 0,Y 446.782,Z 1158.621,A -85,B 0,C 180,E1 14695.447,E2 14695.447} C_VEL
LIN {X 0,Y 444.236,Z 1169.795,A -85,B 0,C 180,E1 14692.218,E2 14692.218} C_VEL
LIN {X 0,Y 442.689,Z 1177.823,A -85,B 0,C 180,E1 14689.528,E2 14689.528} C_VEL
LIN {X 0,Y 441.542,Z 1184.699,A -85,B 0,C 180,E1 14686.849,E2 14686.849} C_VEL
LIN {X 0,Y 440.823,Z 1190.218,A -85,B 0,C 180,E1 14684.314,E2 14684.314} C_VEL
LIN {X 0,Y 440.322,Z 1195.001,A -85,B 0,C 180,E1 14681.659,E2 14681.659} C_VEL
LIN {X 0,Y 440.072,Z 1198.768,A -85,B 0,C 180,E1 14679.019,E2 14679.019} C_VEL
LIN {X 0,Y 439.959,Z 1201.558,A -85,B 0,C 180,E1 14676.393,E2 14676.393} C_VEL
LIN {X 0,Y 439.92,Z 1203.391,A -85,B 0,C 180,E1 14673.779,E2 14673.779} C_VEL
LIN {X 0,Y 439.919,Z 1204.283,A -85,B 0,C 180,E1 14671.172,E2 14671.172} C_VEL
LIN {X 0,Y 439.921,Z 1204.26,A -85,B 0,C 180,E1 14668.697,E2 14668.697} C_VEL
LIN {X 0,Y 439.92,Z 1203.322,A -85,B 0,C 180,E1 14666.09,E2 14666.09} C_VEL
LIN {X 0,Y 439.963,Z 1201.441,A -85,B 0,C 180,E1 14663.475,E2 14663.475} C_VEL
LIN {X 0,Y 440.079,Z 1198.603,A -85,B 0,C 180,E1 14660.848,E2 14660.848} C_VEL
LIN {X 0,Y 440.343,Z 1194.786,A -85,B 0,C 180,E1 14658.208,E2 14658.208} C_VEL
LIN {X 0,Y 440.886,Z 1189.695,A -85,B 0,C 180,E1 14655.42,E2 14655.42} C_VEL
LIN {X 0,Y 441.864,Z 1182.708,A -85,B 0,C 180,E1 14652.304,E2 14652.304} C_VEL
LIN {X 0,Y 443.65,Z 1172.77,A -85,B 0,C 180,E1 14648.724,E2 14648.724} C_VEL
LIN {X 0,Y 445.631,Z 1163.436,A -85,B 0,C 180,E1 14645.898,E2 14645.898} C_VEL
LIN {X 0,Y 448.057,Z 1153.27,A -85,B 0,C 180,E1 14643.206,E2 14643.206} C_VEL
LIN {X 0,Y 451.268,Z 1141.207,A -85,B 0,C 180,E1 14640.389,E2 14640.389} C_VEL
LIN {X 0,Y 455.961,Z 1124.65,A -85,B 0,C 180,E1 14637.054,E2 14637.054} C_VEL
LIN {X 0,Y 460.029,Z 1111.127,A -85,B 0,C 180,E1 14634.679,E2 14634.679} C_VEL
LIN {X 0,Y 464.385,Z 1096.98,A -85,B 0,C 180,E1 14632.458,E2 14632.458} C_VEL
LIN {X 0,Y 469.409,Z 1080.858,A -85,B 0,C 180,E1 14630.201,E2 14630.201} C_VEL
LIN {X 0,Y 476.153,Z 1058.969,A -85,B 0,C 180,E1 14627.536,E2 14627.536} C_VEL
LIN {X 0,Y 481.674,Z 1040.677,A -85,B 0,C 180,E1 14625.608,E2 14625.608} C_VEL
LIN {X 0,Y 487.053,Z 1022.332,A -85,B 0,C 180,E1 14623.898,E2 14623.898} C_VEL
LIN {X 0,Y 493.452,Z 999.62,A -85,B 0,C 180,E1 14622.043,E2 14622.043} C_VEL
LIN {X 0,Y 499.39,Z 976.506,A -85,B 0,C 180,E1 14620.445,E2 14620.445} C_VEL
LIN {X 0,Y 504.233,Z 956.362,A -85,B 0,C 180,E1 14619.241,E2 14619.241} C_VEL
LIN {X 0,Y 508.488,Z 936.956,A -85,B 0,C 180,E1 14618.227,E2 14618.227} C_VEL
LIN {X 0,Y 512.951,Z 914.555,A -85,B 0,C 180,E1 14617.224,E2 14617.224} C_VEL
LIN {X 0,Y 517.704,Z 886.538,A -85,B 0,C 180,E1 14616.204,E2 14616.204} C_VEL
LIN {X 0,Y 520.861,Z 864.072,A -85,B 0,C 180,E1 14615.555,E2 14615.555} C_VEL
LIN {X 0,Y 523.355,Z 842.374,A -85,B 0,C 180,E1 14615.055,E2 14615.055} C_VEL
LIN {X 0,Y 525.463,Z 816.554,A -85,B 0,C 180,E1 14614.588,E2 14614.588} C_VEL
LIN {X 0,Y 537.528,Z 592.335,A -85,B 0,C 180,E1 14611.076,E2 14611.076} C_VEL
LIN {X 0,Y 543.778,Z 478.919,A -85,B 0,C 180,E1 14609.283,E2 14609.283} C_VEL
LIN {X 0,Y 532.054,Z 461.149,A -85,B 0,C 180,E1 14606.659,E2 14606.659} C_VEL
LIN {X 0,Y 521.963,Z 446.927,A -85,B 0,C 180,E1 14604.141,E2 14604.141} C_VEL
LIN {X 0,Y 514.266,Z 436.781,A -85,B 0,C 180,E1 14602.01,E2 14602.01} C_VEL
LIN {X 0,Y 509.505,Z 430.629,A -85,B 0,C 180,E1 14600.566,E2 14600.566} C_VEL
LIN {X 0,Y 506.211,Z 426.424,A -85,B 0,C 180,E1 14599.501,E2 14599.501} C_VEL
LIN {X 0,Y 502.147,Z 421.381,A -85,B 0,C 180,E1 14598.097,E2 14598.097} C_VEL
LIN {X 0,Y 497.919,Z 416.186,A -85,B 0,C 180,E1 14596.508,E2 14596.508} C_VEL
LIN {X 0,Y 493.379,Z 410.794,A -85,B 0,C 180,E1 14594.615,E2 14594.615} C_VEL
LIN {X 0,Y 489.524,Z 406.354,A -85,B 0,C 180,E1 14592.804,E2 14592.804} C_VEL
LIN {X 0,Y 488.077,Z 404.761,A -85,B 0,C 180,E1 14592.062,E2 14592.062} C_VEL
LIN {X 0,Y 483.911,Z 399.972,A -85,B 0,C 180,E1 14589.635,E2 14589.635} C_VEL
LIN {X 0,Y 477.44,Z 393.114,A -85,B 0,C 180,E1 14584.204,E2 14584.204} C_VEL
LIN {X 0,Y 474.87,Z 391.497,A -85,B 0,C 180,E1 14579.517,E2 14579.517} C_VEL
LIN {X 0,Y 475.126,Z 392.098,A -85,B 0,C 180,E1 14575.05,E2 14575.05} C_VEL
LIN {X 0,Y 475.938,Z 393.231,A -85,B 0,C 180,E1 14573.243,E2 14573.243} C_VEL
LIN {X 0,Y 480.196,Z 398.776,A -85,B 0,C 180,E1 14568.408,E2 14568.408} C_VEL
LIN {X 0,Y 484.539,Z 404.535,A -85,B 0,C 180,E1 14565.296,E2 14565.296} C_VEL
LIN {X 0,Y 488.337,Z 409.177,A -85,B 0,C 180,E1 14563.158,E2 14563.158} C_VEL
LIN {X 0,Y 496.409,Z 419.88,A -85,B 0,C 180,E1 14559.452,E2 14559.452} C_VEL
LIN {X 0,Y 501.943,Z 427.547,A -85,B 0,C 180,E1 14557.328,E2 14557.328} C_VEL
LIN {X 0,Y 508.232,Z 436.241,A -85,B 0,C 180,E1 14555.194,E2 14555.194} C_VEL
LIN {X 0,Y 514.112,Z 444.551,A -85,B 0,C 180,E1 14553.397,E2 14553.397} C_VEL
LIN {X 0,Y 522.801,Z 457.342,A -85,B 0,C 180,E1 14550.998,E2 14550.998} C_VEL
LIN {X 0,Y 533.146,Z 473.39,A -85,B 0,C 180,E1 14548.449,E2 14548.449} C_VEL
LIN {X 0,Y 540.472,Z 485.797,A -85,B 0,C 180,E1 14546.789,E2 14546.789} C_VEL
LIN {X 0,Y 528.608,Z 716.907,A -85,B 0,C 180,E1 14543.325,E2 14543.325} C_VEL
LIN {X 0,Y 522.913,Z 831.218,A -85,B 0,C 180,E1 14541.605,E2 14541.605} C_VEL
LIN {X 0,Y 520.36,Z 858.52,A -85,B 0,C 180,E1 14541.063,E2 14541.063} C_VEL
LIN {X 0,Y 517.379,Z 880.985,A -85,B 0,C 180,E1 14540.465,E2 14540.465} C_VEL
LIN {X 0,Y 514.151,Z 901.21,A -85,B 0,C 180,E1 14539.798,E2 14539.798} C_VEL
LIN {X 0,Y 510.069,Z 923.296,A -85,B 0,C 180,E1 14538.915,E2 14538.915} C_VEL
LIN {X 0,Y 504.555,Z 948.831,A -85,B 0,C 180,E1 14537.661,E2 14537.661} C_VEL
LIN {X 0,Y 499.737,Z 968.581,A -85,B 0,C 180,E1 14536.505,E2 14536.505} C_VEL
LIN {X 0,Y 494.63,Z 987.882,A -85,B 0,C 180,E1 14535.197,E2 14535.197} C_VEL
LIN {X 0,Y 487.94,Z 1011.133,A -85,B 0,C 180,E1 14533.352,E2 14533.352} C_VEL
LIN {X 0,Y 482.265,Z 1029.483,A -85,B 0,C 180,E1 14531.644,E2 14531.644} C_VEL
LIN {X 0,Y 476.947,Z 1046.031,A -85,B 0,C 180,E1 14529.888,E2 14529.888} C_VEL
LIN {X 0,Y 470.671,Z 1065.077,A -85,B 0,C 180,E1 14527.568,E2 14527.568} C_VEL
LIN {X 0,Y 464.983,Z 1081.735,A -85,B 0,C 180,E1 14525.191,E2 14525.191} C_VEL
LIN {X 0,Y 460.465,Z 1095.075,A -85,B 0,C 180,E1 14523.027,E2 14523.027} C_VEL
LIN {X 0,Y 455.411,Z 1110.426,A -85,B 0,C 180,E1 14520.184,E2 14520.184} C_VEL
LIN {X 0,Y 451.151,Z 1123.662,A -85,B 0,C 180,E1 14517.284,E2 14517.284} C_VEL
LIN {X 0,Y 449.349,Z 1129.716,A -85,B 0,C 180,E1 14515.824,E2 14515.824} C_VEL
LIN {X 0,Y 447.377,Z 1133.194,A -85,B 0,C 180,E1 14514.971,E2 14514.971} C_VEL
LIN {X 0,Y 438.954,Z 1142.436,A -85,B 0,C 180,E1 14512.748,E2 14512.748} C_VEL
LIN {X 0,Y 437.533,Z 1145.015,A -85,B 0,C 180,E1 14511.968,E2 14511.968} C_VEL
LIN {X 0,Y 435.181,Z 1154.291,A -85,B 0,C 180,E1 14508.625,E2 14508.625} C_VEL
LIN {X 0,Y 433.812,Z 1160.907,A -85,B 0,C 180,E1 14505.782,E2 14505.782} C_VEL
LIN {X 0,Y 432.78,Z 1167.349,A -85,B 0,C 180,E1 14502.408,E2 14502.408} C_VEL
LIN {X 0,Y 432.229,Z 1172.138,A -85,B 0,C 180,E1 14498.96,E2 14498.96} C_VEL
LIN {X 0,Y 432.03,Z 1174.856,A -85,B 0,C 180,E1 14496.245,E2 14496.245} C_VEL
LIN {X 0,Y 431.957,Z 1176.587,A -85,B 0,C 180,E1 14493.584,E2 14493.584} C_VEL
LIN {X 0,Y 431.943,Z 1177.392,A -85,B 0,C 180,E1 14490.929,E2 14490.929} C_VEL
LIN {X 0,Y 431.952,Z 1177.214,A -85,B 0,C 180,E1 14487.878,E2 14487.878} C_VEL
LIN {X 0,Y 431.999,Z 1175.476,A -85,B 0,C 180,E1 14484.422,E2 14484.422} C_VEL
LIN {X 0,Y 432.183,Z 1172.752,A -85,B 0,C 180,E1 14481.485,E2 14481.485} C_VEL
LIN {X 0,Y 432.537,Z 1169.089,A -85,B 0,C 180,E1 14478.668,E2 14478.668} C_VEL
LIN {X 0,Y 433.304,Z 1163.861,A -85,B 0,C 180,E1 14475.569,E2 14475.569} C_VEL
LIN {X 0,Y 434.772,Z 1156.222,A -85,B 0,C 180,E1 14472.051,E2 14472.051} C_VEL
LIN {X 0,Y 436.591,Z 1148.476,A -85,B 0,C 180,E1 14469.134,E2 14469.134} C_VEL
LIN {X 0,Y 439.067,Z 1139.43,A -85,B 0,C 180,E1 14466.23,E2 14466.23} C_VEL
LIN {X 0,Y 443.026,Z 1126.453,A -85,B 0,C 180,E1 14462.732,E2 14462.732} C_VEL
LIN {X 0,Y 446.865,Z 1114.829,A -85,B 0,C 180,E1 14460.068,E2 14460.068} C_VEL
LIN {X 0,Y 451.74,Z 1100.763,A -85,B 0,C 180,E1 14457.257,E2 14457.257} C_VEL
LIN {X 0,Y 457.531,Z 1084.247,A -85,B 0,C 180,E1 14454.458,E2 14454.458} C_VEL
LIN {X 0,Y 462.385,Z 1070.514,A -85,B 0,C 180,E1 14452.425,E2 14452.425} C_VEL
LIN {X 0,Y 467.717,Z 1055.266,A -85,B 0,C 180,E1 14450.427,E2 14450.427} C_VEL
LIN {X 0,Y 474.665,Z 1034.797,A -85,B 0,C 180,E1 14448.106,E2 14448.106} C_VEL
LIN {X 0,Y 480.614,Z 1016.3,A -85,B 0,C 180,E1 14446.315,E2 14446.315} C_VEL
LIN {X 0,Y 486.117,Z 998.346,A -85,B 0,C 180,E1 14444.797,E2 14444.797} C_VEL
LIN {X 0,Y 492.451,Z 976.225,A -85,B 0,C 180,E1 14443.178,E2 14443.178} C_VEL
LIN {X 0,Y 498.165,Z 953.848,A -85,B 0,C 180,E1 14441.811,E2 14441.811} C_VEL
LIN {X 0,Y 502.638,Z 934.643,A -85,B 0,C 180,E1 14440.808,E2 14440.808} C_VEL
LIN {X 0,Y 506.908,Z 914.065,A -85,B 0,C 180,E1 14439.888,E2 14439.888} C_VEL
LIN {X 0,Y 511.534,Z 887.885,A -85,B 0,C 180,E1 14438.938,E2 14438.938} C_VEL
LIN {X 0,Y 514.628,Z 866.143,A -85,B 0,C 180,E1 14438.314,E2 14438.314} C_VEL
LIN {X 0,Y 517.119,Z 844.33,A -85,B 0,C 180,E1 14437.824,E2 14437.824} C_VEL
LIN {X 0,Y 519.181,Z 817.041,A -85,B 0,C 180,E1 14437.355,E2 14437.355} C_VEL
LIN {X 0,Y 531.037,Z 584.628,A -85,B 0,C 180,E1 14433.869,E2 14433.869} C_VEL
LIN {X 0,Y 536.158,Z 489.73,A -85,B 0,C 180,E1 14432.423,E2 14432.423} C_VEL
LIN {X 0,Y 526.173,Z 473.29,A -85,B 0,C 180,E1 14430.049,E2 14430.049} C_VEL
LIN {X 0,Y 516.794,Z 458.931,A -85,B 0,C 180,E1 14427.575,E2 14427.575} C_VEL
LIN {X 0,Y 508.318,Z 446.407,A -85,B 0,C 180,E1 14425.05,E2 14425.05} C_VEL
LIN {X 0,Y 501.505,Z 436.781,A -85,B 0,C 180,E1 14422.755,E2 14422.755} C_VEL
LIN {X 0,Y 497.381,Z 431.176,A -85,B 0,C 180,E1 14421.214,E2 14421.214} C_VEL
LIN {X 0,Y 493.145,Z 425.396,A -85,B 0,C 180,E1 14419.463,E2 14419.463} C_VEL
LIN {X 0,Y 489.605,Z 420.797,A -85,B 0,C 180,E1 14417.839,E2 14417.839} C_VEL
LIN {X 0,Y 486.511,Z 416.449,A -85,B 0,C 180,E1 14416.231,E2 14416.231} C_VEL
LIN {X 0,Y 483.004,Z 411.788,A -85,B 0,C 180,E1 14414.139,E2 14414.139} C_VEL
LIN {X 0,Y 478.399,Z 405.756,A -85,B 0,C 180,E1 14410.599,E2 14410.599} C_VEL
LIN {X 0,Y 474.65,Z 400.47,A -85,B 0,C 180,E1 14405.44,E2 14405.44} C_VEL
LIN {X 0,Y 474.084,Z 399.642,A -85,B 0,C 180,E1 14400.846,E2 14400.846} C_VEL
LIN {X 0,Y 476.31,Z 401.003,A -85,B 0,C 180,E1 14396.269,E2 14396.269} C_VEL
LIN {X 0,Y 478.068,Z 403.306,A -85,B 0,C 180,E1 14394.238,E2 14394.238} C_VEL
LIN {X 0,Y 482.679,Z 407.788,A -85,B 0,C 180,E1 14390.641,E2 14390.641} C_VEL
LIN {X 0,Y 486.845,Z 412.603,A -85,B 0,C 180,E1 14388.148,E2 14388.148} C_VEL
LIN {X 0,Y 488.149,Z 414.105,A -85,B 0,C 180,E1 14387.46,E2 14387.46} C_VEL
LIN {X 0,Y 492.052,Z 418.62,A -85,B 0,C 180,E1 14385.586,E2 14385.586} C_VEL
LIN {X 0,Y 497.918,Z 425.795,A -85,B 0,C 180,E1 14383.131,E2 14383.131} C_VEL
LIN {X 0,Y 502.661,Z 431.734,A -85,B 0,C 180,E1 14381.381,E2 14381.381} C_VEL
LIN {X 0,Y 507.212,Z 437.556,A -85,B 0,C 180,E1 14379.849,E2 14379.849} C_VEL
LIN {X 0,Y 514.104,Z 446.47,A -85,B 0,C 180,E1 14377.742,E2 14377.742} C_VEL
LIN {X 0,Y 524.05,Z 460.21,A -85,B 0,C 180,E1 14375.03,E2 14375.03} C_VEL
LIN {X 0,Y 533.066,Z 473.612,A -85,B 0,C 180,E1 14372.823,E2 14372.823} C_VEL
LIN {X 0,Y 539.507,Z 483.766,A -85,B 0,C 180,E1 14371.359,E2 14371.359} C_VEL
LIN {X 0,Y 527.368,Z 696.274,A -85,B 0,C 180,E1 14368.017,E2 14368.017} C_VEL
LIN {X 0,Y 520.031,Z 826.819,A -85,B 0,C 180,E1 14365.949,E2 14365.949} C_VEL
LIN {X 0,Y 517.349,Z 854.306,A -85,B 0,C 180,E1 14365.404,E2 14365.404} C_VEL
LIN {X 0,Y 513.776,Z 880.189,A -85,B 0,C 180,E1 14364.705,E2 14364.705} C_VEL
LIN {X 0,Y 510.297,Z 901.372,A -85,B 0,C 180,E1 14363.997,E2 14363.997} C_VEL
LIN {X 0,Y 506.472,Z 921.775,A -85,B 0,C 180,E1 14363.181,E2 14363.181} C_VEL
LIN {X 0,Y 501.699,Z 944.449,A -85,B 0,C 180,E1 14362.112,E2 14362.112} C_VEL
LIN {X 0,Y 495.418,Z 970.718,A -85,B 0,C 180,E1 14360.623,E2 14360.623} C_VEL
LIN {X 0,Y 490.361,Z 990.091,A -85,B 0,C 180,E1 14359.334,E2 14359.334} C_VEL
LIN {X 0,Y 485.282,Z 1008.31,A -85,B 0,C 180,E1 14357.96,E2 14357.96} C_VEL
LIN {X 0,Y 479.88,Z 1026.676,A -85,B 0,C 180,E1 14356.395,E2 14356.395} C_VEL
LIN {X 0,Y 473.091,Z 1048.911,A -85,B 0,C 180,E1 14354.223,E2 14354.223} C_VEL
LIN {X 0,Y 466.786,Z 1068.52,A -85,B 0,C 180,E1 14351.986,E2 14351.986} C_VEL
LIN {X 0,Y 461.643,Z 1084.402,A -85,B 0,C 180,E1 14349.937,E2 14349.937} C_VEL
LIN {X 0,Y 456.568,Z 1100.096,A -85,B 0,C 180,E1 14347.662,E2 14347.662} C_VEL
LIN {X 0,Y 450.704,Z 1118.492,A -85,B 0,C 180,E1 14344.606,E2 14344.606} C_VEL
LIN {X 0,Y 446.357,Z 1132.587,A -85,B 0,C 180,E1 14341.896,E2 14341.896} C_VEL
LIN {X 0,Y 442.88,Z 1144.407,A -85,B 0,C 180,E1 14339.335,E2 14339.335} C_VEL
LIN {X 0,Y 439.86,Z 1155.565,A -85,B 0,C 180,E1 14336.603,E2 14336.603} C_VEL
LIN {X 0,Y 436.819,Z 1168.13,A -85,B 0,C 180,E1 14333.042,E2 14333.042} C_VEL
LIN {X 0,Y 434.94,Z 1177.087,A -85,B 0,C 180,E1 14330.031,E2 14330.031} C_VEL
LIN {X 0,Y 433.712,Z 1184.041,A -85,B 0,C 180,E1 14327.301,E2 14327.301} C_VEL
LIN {X 0,Y 432.883,Z 1189.897,A -85,B 0,C 180,E1 14324.582,E2 14324.582} C_VEL
LIN {X 0,Y 432.355,Z 1194.703,A -85,B 0,C 180,E1 14321.877,E2 14321.877} C_VEL
LIN {X 0,Y 432.083,Z 1198.494,A -85,B 0,C 180,E1 14319.188,E2 14319.188} C_VEL
LIN {X 0,Y 431.964,Z 1201.299,A -85,B 0,C 180,E1 14316.512,E2 14316.512} C_VEL
LIN {X 0,Y 431.923,Z 1203.147,A -85,B 0,C 180,E1 14313.837,E2 14313.837} C_VEL
LIN {X 0,Y 431.923,Z 1204.036,A -85,B 0,C 180,E1 14311.194,E2 14311.194} C_VEL
LIN {X 0,Y 431.924,Z 1204.012,A -85,B 0,C 180,E1 14308.673,E2 14308.673} C_VEL
LIN {X 0,Y 431.923,Z 1203.14,A -85,B 0,C 180,E1 14306.15,E2 14306.15} C_VEL
LIN {X 0,Y 431.965,Z 1201.298,A -85,B 0,C 180,E1 14303.487,E2 14303.487} C_VEL
LIN {X 0,Y 432.082,Z 1198.496,A -85,B 0,C 180,E1 14300.812,E2 14300.812} C_VEL
LIN {X 0,Y 432.355,Z 1194.711,A -85,B 0,C 180,E1 14298.122,E2 14298.122} C_VEL
LIN {X 0,Y 432.884,Z 1189.912,A -85,B 0,C 180,E1 14295.418,E2 14295.418} C_VEL
LIN {X 0,Y 433.763,Z 1183.733,A -85,B 0,C 180,E1 14292.562,E2 14292.562} C_VEL
LIN {X 0,Y 435.394,Z 1174.868,A -85,B 0,C 180,E1 14289.148,E2 14289.148} C_VEL
LIN {X 0,Y 437.792,Z 1163.855,A -85,B 0,C 180,E1 14285.685,E2 14285.685} C_VEL
LIN {X 0,Y 440.268,Z 1153.964,A -85,B 0,C 180,E1 14282.985,E2 14282.985} C_VEL
LIN {X 0,Y 443.228,Z 1143.22,A -85,B 0,C 180,E1 14280.393,E2 14280.393} C_VEL
LIN {X 0,Y 447.387,Z 1129.213,A -85,B 0,C 180,E1 14277.41,E2 14277.41} C_VEL
LIN {X 0,Y 452.638,Z 1112.335,A -85,B 0,C 180,E1 14274.325,E2 14274.325} C_VEL
LIN {X 0,Y 457.413,Z 1097.463,A -85,B 0,C 180,E1 14271.943,E2 14271.943} C_VEL
LIN {X 0,Y 462.365,Z 1082.18,A -85,B 0,C 180,E1 14269.764,E2 14269.764} C_VEL
LIN {X 0,Y 468.753,Z 1062.529,A -85,B 0,C 180,E1 14267.288,E2 14267.288} C_VEL
LIN {X 0,Y 475.309,Z 1041.48,A -85,B 0,C 180,E1 14265.023,E2 14265.023} C_VEL
LIN {X 0,Y 480.86,Z 1023.234,A -85,B 0,C 180,E1 14263.3,E2 14263.3} C_VEL
LIN {X 0,Y 486.793,Z 1002.911,A -85,B 0,C 180,E1 14261.612,E2 14261.612} C_VEL
LIN {X 0,Y 493.531,Z 977.947,A -85,B 0,C 180,E1 14259.839,E2 14259.839} C_VEL
LIN {X 0,Y 498.739,Z 956.987,A -85,B 0,C 180,E1 14258.573,E2 14258.573} C_VEL
LIN {X 0,Y 503.171,Z 937.433,A -85,B 0,C 180,E1 14257.545,E2 14257.545} C_VEL
LIN {X 0,Y 507.495,Z 916.409,A -85,B 0,C 180,E1 14256.595,E2 14256.595} C_VEL
LIN {X 0,Y 512.377,Z 889.087,A -85,B 0,C 180,E1 14255.577,E2 14255.577} C_VEL
LIN {X 0,Y 515.878,Z 864.995,A -85,B 0,C 180,E1 14254.87,E2 14254.87} C_VEL
LIN {X 0,Y 518.469,Z 843.183,A -85,B 0,C 180,E1 14254.364,E2 14254.364} C_VEL
LIN {X 0,Y 520.524,Z 819.198,A -85,B 0,C 180,E1 14253.924,E2 14253.924} C_VEL
LIN {X 0,Y 532.822,Z 598.462,A -85,B 0,C 180,E1 14250.45,E2 14250.45} C_VEL
LIN {X 0,Y 539.395,Z 483.483,A -85,B 0,C 180,E1 14248.633,E2 14248.633} C_VEL
LIN {X 0,Y 529.16,Z 467.728,A -85,B 0,C 180,E1 14246.272,E2 14246.272} C_VEL
LIN {X 0,Y 519.413,Z 453.797,A -85,B 0,C 180,E1 14243.785,E2 14243.785} C_VEL
LIN {X 0,Y 511.84,Z 443.679,A -85,B 0,C 180,E1 14241.637,E2 14241.637} C_VEL
LIN {X 0,Y 505.221,Z 434.858,A -85,B 0,C 180,E1 14239.54,E2 14239.54} C_VEL
LIN {X 0,Y 499.942,Z 428.406,A -85,B 0,C 180,E1 14237.698,E2 14237.698} C_VEL
LIN {X 0,Y 496.081,Z 423.584,A -85,B 0,C 180,E1 14236.21,E2 14236.21} C_VEL
LIN {X 0,Y 491.75,Z 418.366,A -85,B 0,C 180,E1 14234.363,E2 14234.363} C_VEL
LIN {X 0,Y 487.972,Z 413.884,A -85,B 0,C 180,E1 14232.545,E2 14232.545} C_VEL
LIN {X 0,Y 485.476,Z 411.375,A -85,B 0,C 180,E1 14231.223,E2 14231.223} C_VEL
LIN {X 0,Y 482.045,Z 407.067,A -85,B 0,C 180,E1 14229.07,E2 14229.07} C_VEL
LIN {X 0,Y 476.36,Z 401,A -85,B 0,C 180,E1 14224.093,E2 14224.093} C_VEL
LIN {X 0,Y 473.864,Z 399.429,A -85,B 0,C 180,E1 14219.395,E2 14219.395} C_VEL
LIN {X 0,Y 474.197,Z 400.089,A -85,B 0,C 180,E1 14214.919,E2 14214.919} C_VEL
LIN {X 0,Y 474.899,Z 401.114,A -85,B 0,C 180,E1 14213.35,E2 14213.35} C_VEL
LIN {X 0,Y 479.085,Z 406.71,A -85,B 0,C 180,E1 14208.503,E2 14208.503} C_VEL
LIN {X 0,Y 483.289,Z 412.397,A -85,B 0,C 180,E1 14205.441,E2 14205.441} C_VEL
LIN {X 0,Y 487.463,Z 417.767,A -85,B 0,C 180,E1 14203.066,E2 14203.066} C_VEL
LIN {X 0,Y 494.632,Z 427.262,A -85,B 0,C 180,E1 14199.746,E2 14199.746} C_VEL
LIN {X 0,Y 500.147,Z 435.032,A -85,B 0,C 180,E1 14197.583,E2 14197.583} C_VEL
LIN {X 0,Y 506.269,Z 443.644,A -85,B 0,C 180,E1 14195.465,E2 14195.465} C_VEL
LIN {X 0,Y 511.916,Z 451.748,A -85,B 0,C 180,E1 14193.705,E2 14193.705} C_VEL
LIN {X 0,Y 520.373,Z 464.401,A -85,B 0,C 180,E1 14191.322,E2 14191.322} C_VEL
LIN {X 0,Y 530.272,Z 479.98,A -85,B 0,C 180,E1 14188.828,E2 14188.828} C_VEL
LIN {X 0,Y 536.136,Z 490.053,A -85,B 0,C 180,E1 14187.459,E2 14187.459} C_VEL
LIN {X 0,Y 523.839,Z 721.811,A -85,B 0,C 180,E1 14183.974,E2 14183.974} C_VEL
LIN {X 0,Y 518.188,Z 831.219,A -85,B 0,C 180,E1 14182.319,E2 14182.319} C_VEL
LIN {X 0,Y 515.562,Z 858.539,A -85,B 0,C 180,E1 14181.776,E2 14181.776} C_VEL
LIN {X 0,Y 512.501,Z 880.977,A -85,B 0,C 180,E1 14181.179,E2 14181.179} C_VEL
LIN {X 0,Y 509.174,Z 901.25,A -85,B 0,C 180,E1 14180.511,E2 14180.511} C_VEL
LIN {X 0,Y 504.854,Z 923.997,A -85,B 0,C 180,E1 14179.598,E2 14179.598} C_VEL
LIN {X 0,Y 499.181,Z 949.393,A -85,B 0,C 180,E1 14178.343,E2 14178.343} C_VEL
LIN {X 0,Y 494.158,Z 969.354,A -85,B 0,C 180,E1 14177.166,E2 14177.166} C_VEL
LIN {X 0,Y 488.667,Z 989.439,A -85,B 0,C 180,E1 14175.792,E2 14175.792} C_VEL
LIN {X 0,Y 481.742,Z 1012.542,A -85,B 0,C 180,E1 14173.927,E2 14173.927} C_VEL
LIN {X 0,Y 476.002,Z 1030.473,A -85,B 0,C 180,E1 14172.236,E2 14172.236} C_VEL
LIN {X 0,Y 470.195,Z 1047.924,A -85,B 0,C 180,E1 14170.355,E2 14170.355} C_VEL
LIN {X 0,Y 463.525,Z 1067.229,A -85,B 0,C 180,E1 14167.936,E2 14167.936} C_VEL
LIN {X 0,Y 458.115,Z 1082.521,A -85,B 0,C 180,E1 14165.714,E2 14165.714} C_VEL
LIN {X 0,Y 453.311,Z 1096.149,A -85,B 0,C 180,E1 14163.465,E2 14163.465} C_VEL
LIN {X 0,Y 447.842,Z 1111.965,A -85,B 0,C 180,E1 14160.452,E2 14160.452} C_VEL
LIN {X 0,Y 443.856,Z 1123.87,A -85,B 0,C 180,E1 14157.795,E2 14157.795} C_VEL
LIN {X 0,Y 440.511,Z 1134.474,A -85,B 0,C 180,E1 14155.086,E2 14155.086} C_VEL
LIN {X 0,Y 437.533,Z 1145.015,A -85,B 0,C 180,E1 14151.968,E2 14151.968} C_VEL
LIN {X 0,Y 435.811,Z 1147.935,A -85,B 0,C 180,E1 14151.048,E2 14151.048} C_VEL
LIN {X 0,Y 427.965,Z 1155.358,A -85,B 0,C 180,E1 14148.618,E2 14148.618} C_VEL
LIN {X 0,Y 426.765,Z 1157.489,A -85,B 0,C 180,E1 14147.788,E2 14147.788} C_VEL
LIN {X 0,Y 425.305,Z 1164.687,A -85,B 0,C 180,E1 14144.292,E2 14144.292} C_VEL
LIN {X 0,Y 424.58,Z 1169.409,A -85,B 0,C 180,E1 14141.41,E2 14141.41} C_VEL
LIN {X 0,Y 424.205,Z 1173.052,A -85,B 0,C 180,E1 14138.54,E2 14138.54} C_VEL
LIN {X 0,Y 424.004,Z 1175.867,A -85,B 0,C 180,E1 14135.413,E2 14135.413} C_VEL
LIN {X 0,Y 423.95,Z 1177.489,A -85,B 0,C 180,E1 14131.892,E2 14131.892} C_VEL
LIN {X 0,Y 423.948,Z 1177.654,A -85,B 0,C 180,E1 14129.054,E2 14129.054} C_VEL
LIN {X 0,Y 423.957,Z 1176.881,A -85,B 0,C 180,E1 14126.349,E2 14126.349} C_VEL
LIN {X 0,Y 424.042,Z 1175.183,A -85,B 0,C 180,E1 14123.637,E2 14123.637} C_VEL
LIN {X 0,Y 424.255,Z 1172.396,A -85,B 0,C 180,E1 14120.778,E2 14120.778} C_VEL
LIN {X 0,Y 424.835,Z 1167.766,A -85,B 0,C 180,E1 14117.357,E2 14117.357} C_VEL
LIN {X 0,Y 425.924,Z 1161.374,A -85,B 0,C 180,E1 14113.918,E2 14113.918} C_VEL
LIN {X 0,Y 427.361,Z 1154.796,A -85,B 0,C 180,E1 14111.022,E2 14111.022} C_VEL
LIN {X 0,Y 429.631,Z 1146.226,A -85,B 0,C 180,E1 14107.851,E2 14107.851} C_VEL
LIN {X 0,Y 432.988,Z 1134.983,A -85,B 0,C 180,E1 14104.417,E2 14104.417} C_VEL
LIN {X 0,Y 436.448,Z 1124.525,A -85,B 0,C 180,E1 14101.691,E2 14101.691} C_VEL
LIN {X 0,Y 440.833,Z 1112.049,A -85,B 0,C 180,E1 14098.86,E2 14098.86} C_VEL
LIN {X 0,Y 446.571,Z 1096.201,A -85,B 0,C 180,E1 14095.807,E2 14095.807} C_VEL
LIN {X 0,Y 451.452,Z 1082.924,A -85,B 0,C 180,E1 14093.59,E2 14093.59} C_VEL
LIN {X 0,Y 457.041,Z 1067.725,A -85,B 0,C 180,E1 14091.355,E2 14091.355} C_VEL
LIN {X 0,Y 464.353,Z 1047.342,A -85,B 0,C 180,E1 14088.784,E2 14088.784} C_VEL
LIN {X 0,Y 470.192,Z 1030.409,A -85,B 0,C 180,E1 14086.952,E2 14086.952} C_VEL
LIN {X 0,Y 476.035,Z 1012.769,A -85,B 0,C 180,E1 14085.28,E2 14085.28} C_VEL
LIN {X 0,Y 483.359,Z 989.084,A -85,B 0,C 180,E1 14083.364,E2 14083.364} C_VEL
LIN {X 0,Y 488.761,Z 969.906,A -85,B 0,C 180,E1 14082.047,E2 14082.047} C_VEL
LIN {X 0,Y 493.893,Z 950.135,A -85,B 0,C 180,E1 14080.875,E2 14080.875} C_VEL
LIN {X 0,Y 499.482,Z 926.202,A -85,B 0,C 180,E1 14079.673,E2 14079.673} C_VEL
LIN {X 0,Y 504.169,Z 902.313,A -85,B 0,C 180,E1 14078.704,E2 14078.704} C_VEL
LIN {X 0,Y 507.721,Z 881.35,A -85,B 0,C 180,E1 14078.009,E2 14078.009} C_VEL
LIN {X 0,Y 510.784,Z 859.555,A -85,B 0,C 180,E1 14077.426,E2 14077.426} C_VEL
LIN {X 0,Y 513.593,Z 831.645,A -85,B 0,C 180,E1 14076.865,E2 14076.865} C_VEL
LIN {X 0,Y 518.283,Z 744.582,A -85,B 0,C 180,E1 14075.538,E2 14075.538} C_VEL
LIN {X 0,Y 530.484,Z 520.003,A -85,B 0,C 180,E1 14072.149,E2 14072.149} C_VEL
LIN {X 0,Y 531.959,Z 494.153,A -85,B 0,C 180,E1 14071.756,E2 14071.756} C_VEL
LIN {X 0,Y 522.811,Z 479.005,A -85,B 0,C 180,E1 14069.51,E2 14069.51} C_VEL
LIN {X 0,Y 514.162,Z 465.56,A -85,B 0,C 180,E1 14067.163,E2 14067.163} C_VEL
LIN {X 0,Y 506.009,Z 453.35,A -85,B 0,C 180,E1 14064.673,E2 14064.673} C_VEL
LIN {X 0,Y 499.628,Z 444.156,A -85,B 0,C 180,E1 14062.473,E2 14062.473} C_VEL
LIN {X 0,Y 495.49,Z 438.453,A -85,B 0,C 180,E1 14060.891,E2 14060.891} C_VEL
LIN {X 0,Y 491.326,Z 432.679,A -85,B 0,C 180,E1 14059.126,E2 14059.126} C_VEL
LIN {X 0,Y 487.829,Z 428.059,A -85,B 0,C 180,E1 14057.474,E2 14057.474} C_VEL
LIN {X 0,Y 485.019,Z 424.047,A -85,B 0,C 180,E1 14055.975,E2 14055.975} C_VEL
LIN {X 0,Y 480.974,Z 418.712,A -85,B 0,C 180,E1 14053.464,E2 14053.464} C_VEL
LIN {X 0,Y 477.305,Z 413.639,A -85,B 0,C 180,E1 14050.501,E2 14050.501} C_VEL
LIN {X 0,Y 473.631,Z 408.371,A -85,B 0,C 180,E1 14045.33,E2 14045.33} C_VEL
LIN {X 0,Y 473.106,Z 407.582,A -85,B 0,C 180,E1 14040.848,E2 14040.848} C_VEL
LIN {X 0,Y 475.331,Z 408.957,A -85,B 0,C 180,E1 14036.261,E2 14036.261} C_VEL
LIN {X 0,Y 481.427,Z 415.605,A -85,B 0,C 180,E1 14030.797,E2 14030.797} C_VEL
LIN {X 0,Y 485.647,Z 420.485,A -85,B 0,C 180,E1 14028.239,E2 14028.239} C_VEL
LIN {X 0,Y 487.355,Z 422.767,A -85,B 0,C 180,E1 14027.319,E2 14027.319} C_VEL
LIN {X 0,Y 491.55,Z 427.586,A -85,B 0,C 180,E1 14025.33,E2 14025.33} C_VEL
LIN {X 0,Y 496.209,Z 433.338,A -85,B 0,C 180,E1 14023.373,E2 14023.373} C_VEL
LIN {X 0,Y 501.039,Z 439.492,A -85,B 0,C 180,E1 14021.56,E2 14021.56} C_VEL
LIN {X 0,Y 505.219,Z 444.903,A -85,B 0,C 180,E1 14020.128,E2 14020.128} C_VEL
LIN {X 0,Y 512.016,Z 453.856,A -85,B 0,C 180,E1 14018.009,E2 14018.009} C_VEL
LIN {X 0,Y 521.557,Z 467.209,A -85,B 0,C 180,E1 14015.356,E2 14015.356} C_VEL
LIN {X 0,Y 530.552,Z 480.8,A -85,B 0,C 180,E1 14013.108,E2 14013.108} C_VEL
LIN {X 0,Y 535.175,Z 488.165,A -85,B 0,C 180,E1 14012.029,E2 14012.029} C_VEL
LIN {X 0,Y 522.696,Z 700.187,A -85,B 0,C 180,E1 14008.685,E2 14008.685} C_VEL
LIN {X 0,Y 515.347,Z 826.879,A -85,B 0,C 180,E1 14006.67,E2 14006.67} C_VEL
LIN {X 0,Y 512.589,Z 854.425,A -85,B 0,C 180,E1 14006.123,E2 14006.123} C_VEL
LIN {X 0,Y 508.946,Z 880.172,A -85,B 0,C 180,E1 14005.428,E2 14005.428} C_VEL
LIN {X 0,Y 505.284,Z 901.841,A -85,B 0,C 180,E1 14004.702,E2 14004.702} C_VEL
LIN {X 0,Y 501.058,Z 923.652,A -85,B 0,C 180,E1 14003.822,E2 14003.822} C_VEL
LIN {X 0,Y 495.145,Z 950.322,A -85,B 0,C 180,E1 14002.524,E2 14002.524} C_VEL
LIN {X 0,Y 489.707,Z 972.009,A -85,B 0,C 180,E1 14001.257,E2 14001.257} C_VEL
LIN {X 0,Y 484.508,Z 991.242,A -85,B 0,C 180,E1 13999.963,E2 13999.963} C_VEL
LIN {X 0,Y 479.374,Z 1009.014,A -85,B 0,C 180,E1 13998.608,E2 13998.608} C_VEL
LIN {X 0,Y 473.294,Z 1029.001,A -85,B 0,C 180,E1 13996.878,E2 13996.878} C_VEL
LIN {X 0,Y 465.916,Z 1051.959,A -85,B 0,C 180,E1 13994.561,E2 13994.561} C_VEL
LIN {X 0,Y 460.187,Z 1069.178,A -85,B 0,C 180,E1 13992.559,E2 13992.559} C_VEL
LIN {X 0,Y 454.847,Z 1085.034,A -85,B 0,C 180,E1 13990.481,E2 13990.481} C_VEL
LIN {X 0,Y 449.034,Z 1102.334,A -85,B 0,C 180,E1 13987.921,E2 13987.921} C_VEL
LIN {X 0,Y 443.261,Z 1119.585,A -85,B 0,C 180,E1 13984.956,E2 13984.956} C_VEL
LIN {X 0,Y 439.008,Z 1132.814,A -85,B 0,C 180,E1 13982.359,E2 13982.359} C_VEL
LIN {X 0,Y 435.364,Z 1144.654,A -85,B 0,C 180,E1 13979.74,E2 13979.74} C_VEL
LIN {X 0,Y 431.799,Z 1157.357,A -85,B 0,C 180,E1 13976.545,E2 13976.545} C_VEL
LIN {X 0,Y 428.817,Z 1169.054,A -85,B 0,C 180,E1 13973.062,E2 13973.062} C_VEL
LIN {X 0,Y 426.971,Z 1177.552,A -85,B 0,C 180,E1 13970.103,E2 13970.103} C_VEL
LIN {X 0,Y 425.672,Z 1184.655,A -85,B 0,C 180,E1 13967.215,E2 13967.215} C_VEL
LIN {X 0,Y 424.817,Z 1190.647,A -85,B 0,C 180,E1 13964.308,E2 13964.308} C_VEL
LIN {X 0,Y 424.215,Z 1196.55,A -85,B 0,C 180,E1 13960.731,E2 13960.731} C_VEL
LIN {X 0,Y 423.996,Z 1200.444,A -85,B 0,C 180,E1 13957.316,E2 13957.316} C_VEL
LIN {X 0,Y 423.93,Z 1202.604,A -85,B 0,C 180,E1 13954.464,E2 13954.464} C_VEL
LIN {X 0,Y 423.922,Z 1203.693,A -85,B 0,C 180,E1 13951.757,E2 13951.757} C_VEL
LIN {X 0,Y 423.921,Z 1203.835,A -85,B 0,C 180,E1 13949.054,E2 13949.054} C_VEL
LIN {X 0,Y 423.926,Z 1203.03,A -85,B 0,C 180,E1 13946.349,E2 13946.349} C_VEL
LIN {X 0,Y 423.966,Z 1201.157,A -85,B 0,C 180,E1 13943.5,E2 13943.5} C_VEL
LIN {X 0,Y 424.084,Z 1198.39,A -85,B 0,C 180,E1 13940.774,E2 13940.774} C_VEL
LIN {X 0,Y 424.368,Z 1194.634,A -85,B 0,C 180,E1 13938.033,E2 13938.033} C_VEL
LIN {X 0,Y 424.915,Z 1189.849,A -85,B 0,C 180,E1 13935.274,E2 13935.274} C_VEL
LIN {X 0,Y 425.804,Z 1183.862,A -85,B 0,C 180,E1 13932.438,E2 13932.438} C_VEL
LIN {X 0,Y 427.23,Z 1176.281,A -85,B 0,C 180,E1 13929.417,E2 13929.417} C_VEL
LIN {X 0,Y 429.786,Z 1165.071,A -85,B 0,C 180,E1 13925.683,E2 13925.683} C_VEL
LIN {X 0,Y 432.634,Z 1154.153,A -85,B 0,C 180,E1 13922.618,E2 13922.618} C_VEL
LIN {X 0,Y 435.728,Z 1143.465,A -85,B 0,C 180,E1 13919.983,E2 13919.983} C_VEL
LIN {X 0,Y 439.625,Z 1130.834,A -85,B 0,C 180,E1 13917.227,E2 13917.227} C_VEL
LIN {X 0,Y 445.32,Z 1113.391,A -85,B 0,C 180,E1 13913.932,E2 13913.932} C_VEL
LIN {X 0,Y 450.479,Z 1097.957,A -85,B 0,C 180,E1 13911.413,E2 13911.413} C_VEL
LIN {X 0,Y 455.585,Z 1082.818,A -85,B 0,C 180,E1 13909.217,E2 13909.217} C_VEL
LIN {X 0,Y 461.314,Z 1065.823,A -85,B 0,C 180,E1 13907.03,E2 13907.03} C_VEL
LIN {X 0,Y 468.61,Z 1043.539,A -85,B 0,C 180,E1 13904.548,E2 13904.548} C_VEL
LIN {X 0,Y 474.305,Z 1025.511,A -85,B 0,C 180,E1 13902.809,E2 13902.809} C_VEL
LIN {X 0,Y 479.945,Z 1006.931,A -85,B 0,C 180,E1 13901.229,E2 13901.229} C_VEL
LIN {X 0,Y 485.432,Z 987.833,A -85,B 0,C 180,E1 13899.799,E2 13899.799} C_VEL
LIN {X 0,Y 491.923,Z 963.473,A -85,B 0,C 180,E1 13898.224,E2 13898.224} C_VEL
LIN {X 0,Y 497.411,Z 940.209,A -85,B 0,C 180,E1 13896.961,E2 13896.961} C_VEL
LIN {X 0,Y 501.905,Z 919.236,A -85,B 0,C 180,E1 13895.994,E2 13895.994} C_VEL
LIN {X 0,Y 505.986,Z 897.723,A -85,B 0,C 180,E1 13895.153,E2 13895.153} C_VEL
LIN {X 0,Y 510.462,Z 869.795,A -85,B 0,C 180,E1 13894.274,E2 13894.274} C_VEL
LIN {X 0,Y 513.495,Z 845.561,A -85,B 0,C 180,E1 13893.692,E2 13893.692} C_VEL
LIN {X 0,Y 515.571,Z 823.027,A -85,B 0,C 180,E1 13893.268,E2 13893.268} C_VEL
LIN {X 0,Y 527.906,Z 609.246,A -85,B 0,C 180,E1 13889.885,E2 13889.885} C_VEL
LIN {X 0,Y 535.093,Z 487.973,A -85,B 0,C 180,E1 13887.971,E2 13887.971} C_VEL
LIN {X 0,Y 525.581,Z 473.309,A -85,B 0,C 180,E1 13885.706,E2 13885.706} C_VEL
LIN {X 0,Y 516.886,Z 460.666,A -85,B 0,C 180,E1 13883.424,E2 13883.424} C_VEL
LIN {X 0,Y 509.437,Z 450.574,A -85,B 0,C 180,E1 13881.261,E2 13881.261} C_VEL
LIN {X 0,Y 502.928,Z 441.855,A -85,B 0,C 180,E1 13879.15,E2 13879.15} C_VEL
LIN {X 0,Y 498.203,Z 435.935,A -85,B 0,C 180,E1 13877.46,E2 13877.46} C_VEL
LIN {X 0,Y 494.397,Z 431.122,A -85,B 0,C 180,E1 13875.965,E2 13875.965} C_VEL
LIN {X 0,Y 490.131,Z 425.934,A -85,B 0,C 180,E1 13874.11,E2 13874.11} C_VEL
LIN {X 0,Y 486.327,Z 421.241,A -85,B 0,C 180,E1 13872.226,E2 13872.226} C_VEL
LIN {X 0,Y 481.314,Z 415.467,A -85,B 0,C 180,E1 13869.265,E2 13869.265} C_VEL
LIN {X 0,Y 475.282,Z 408.887,A -85,B 0,C 180,E1 13863.981,E2 13863.981} C_VEL
LIN {X 0,Y 472.859,Z 407.363,A -85,B 0,C 180,E1 13859.273,E2 13859.273} C_VEL
LIN {X 0,Y 473.319,Z 408.123,A -85,B 0,C 180,E1 13854.667,E2 13854.667} C_VEL
LIN {X 0,Y 474.047,Z 409.4,A -85,B 0,C 180,E1 13853.095,E2 13853.095} C_VEL
LIN {X 0,Y 477.907,Z 414.529,A -85,B 0,C 180,E1 13848.658,E2 13848.658} C_VEL
LIN {X 0,Y 481.956,Z 420.105,A -85,B 0,C 180,E1 13845.645,E2 13845.645} C_VEL
LIN {X 0,Y 486.054,Z 425.505,A -85,B 0,C 180,E1 13843.262,E2 13843.262} C_VEL
LIN {X 0,Y 492.929,Z 434.753,A -85,B 0,C 180,E1 13840.014,E2 13840.014} C_VEL
LIN {X 0,Y 498.434,Z 442.62,A -85,B 0,C 180,E1 13837.812,E2 13837.812} C_VEL
LIN {X 0,Y 504.239,Z 450.923,A -85,B 0,C 180,E1 13835.765,E2 13835.765} C_VEL
LIN {X 0,Y 509.614,Z 458.754,A -85,B 0,C 180,E1 13834.053,E2 13834.053} C_VEL
LIN {X 0,Y 517.866,Z 471.303,A -85,B 0,C 180,E1 13831.674,E2 13831.674} C_VEL
LIN {X 0,Y 527.525,Z 486.737,A -85,B 0,C 180,E1 13829.187,E2 13829.187} C_VEL
LIN {X 0,Y 531.865,Z 494.43,A -85,B 0,C 180,E1 13828.14,E2 13828.14} C_VEL
LIN {X 0,Y 519.163,Z 726.257,A -85,B 0,C 180,E1 13824.642,E2 13824.642} C_VEL
LIN {X 0,Y 513.54,Z 831.288,A -85,B 0,C 180,E1 13823.045,E2 13823.045} C_VEL
LIN {X 0,Y 510.806,Z 858.839,A -85,B 0,C 180,E1 13822.496,E2 13822.496} C_VEL
LIN {X 0,Y 507.691,Z 881.052,A -85,B 0,C 180,E1 13821.905,E2 13821.905} C_VEL
LIN {X 0,Y 504.145,Z 902.049,A -85,B 0,C 180,E1 13821.21,E2 13821.21} C_VEL
LIN {X 0,Y 499.463,Z 925.964,A -85,B 0,C 180,E1 13820.24,E2 13820.24} C_VEL
LIN {X 0,Y 493.878,Z 949.948,A -85,B 0,C 180,E1 13819.039,E2 13819.039} C_VEL
LIN {X 0,Y 488.818,Z 969.484,A -85,B 0,C 180,E1 13817.883,E2 13817.883} C_VEL
LIN {X 0,Y 483.147,Z 989.626,A -85,B 0,C 180,E1 13816.499,E2 13816.499} C_VEL
LIN {X 0,Y 476.133,Z 1012.306,A -85,B 0,C 180,E1 13814.664,E2 13814.664} C_VEL
LIN {X 0,Y 470.317,Z 1029.911,A -85,B 0,C 180,E1 13813.001,E2 13813.001} C_VEL
LIN {X 0,Y 464.549,Z 1046.666,A -85,B 0,C 180,E1 13811.195,E2 13811.195} C_VEL
LIN {X 0,Y 457.743,Z 1065.762,A -85,B 0,C 180,E1 13808.823,E2 13808.823} C_VEL
LIN {X 0,Y 451.92,Z 1081.576,A -85,B 0,C 180,E1 13806.525,E2 13806.525} C_VEL
LIN {X 0,Y 446.988,Z 1094.971,A -85,B 0,C 180,E1 13804.313,E2 13804.313} C_VEL
LIN {X 0,Y 441.902,Z 1109.049,A -85,B 0,C 180,E1 13801.664,E2 13801.664} C_VEL
LIN {X 0,Y 436.805,Z 1123.453,A -85,B 0,C 180,E1 13798.476,E2 13798.476} C_VEL
LIN {X 0,Y 433.243,Z 1134.163,A -85,B 0,C 180,E1 13795.715,E2 13795.715} C_VEL
LIN {X 0,Y 429.944,Z 1145.174,A -85,B 0,C 180,E1 13792.421,E2 13792.421} C_VEL
LIN {X 0,Y 427.492,Z 1154.259,A -85,B 0,C 180,E1 13789.1,E2 13789.1} C_VEL
LIN {X 0,Y 426.765,Z 1157.489,A -85,B 0,C 180,E1 13787.788,E2 13787.788} C_VEL
LIN {X 0,Y 425.295,Z 1159.859,A -85,B 0,C 180,E1 13786.814,E2 13786.814} C_VEL
LIN {X 0,Y 417.907,Z 1165.651,A -85,B 0,C 180,E1 13784.134,E2 13784.134} C_VEL
LIN {X 0,Y 417.04,Z 1167.11,A -85,B 0,C 180,E1 13783.326,E2 13783.326} C_VEL
LIN {X 0,Y 416.319,Z 1172.392,A -85,B 0,C 180,E1 13779.539,E2 13779.539} C_VEL
LIN {X 0,Y 416.068,Z 1175.25,A -85,B 0,C 180,E1 13776.624,E2 13776.624} C_VEL
LIN {X 0,Y 415.973,Z 1177.019,A -85,B 0,C 180,E1 13773.859,E2 13773.859} C_VEL
LIN {X 0,Y 415.955,Z 1177.864,A -85,B 0,C 180,E1 13771.102,E2 13771.102} C_VEL
LIN {X 0,Y 415.956,Z 1177.772,A -85,B 0,C 180,E1 13768.21,E2 13768.21} C_VEL
LIN {X 0,Y 416.005,Z 1176.408,A -85,B 0,C 180,E1 13764.76,E2 13764.76} C_VEL
LIN {X 0,Y 416.219,Z 1173.411,A -85,B 0,C 180,E1 13761.295,E2 13761.295} C_VEL
LIN {X 0,Y 416.619,Z 1169.801,A -85,B 0,C 180,E1 13758.37,E2 13758.37} C_VEL
LIN {X 0,Y 417.388,Z 1165.103,A -85,B 0,C 180,E1 13755.426,E2 13755.426} C_VEL
LIN {X 0,Y 418.973,Z 1157.768,A -85,B 0,C 180,E1 13751.776,E2 13751.776} C_VEL
LIN {X 0,Y 421.083,Z 1149.623,A -85,B 0,C 180,E1 13748.551,E2 13748.551} C_VEL
LIN {X 0,Y 423.581,Z 1141.319,A -85,B 0,C 180,E1 13745.749,E2 13745.749} C_VEL
LIN {X 0,Y 427.285,Z 1130.289,A -85,B 0,C 180,E1 13742.549,E2 13742.549} C_VEL
LIN {X 0,Y 431.936,Z 1117.274,A -85,B 0,C 180,E1 13739.385,E2 13739.385} C_VEL
LIN {X 0,Y 436.505,Z 1105.025,A -85,B 0,C 180,E1 13736.807,E2 13736.807} C_VEL
LIN {X 0,Y 442.086,Z 1090.512,A -85,B 0,C 180,E1 13734.142,E2 13734.142} C_VEL
LIN {X 0,Y 448.779,Z 1072.99,A -85,B 0,C 180,E1 13731.403,E2 13731.403} C_VEL
LIN {X 0,Y 454.443,Z 1057.94,A -85,B 0,C 180,E1 13729.363,E2 13729.363} C_VEL
LIN {X 0,Y 460.209,Z 1042.264,A -85,B 0,C 180,E1 13727.492,E2 13727.492} C_VEL
LIN {X 0,Y 467.433,Z 1021.836,A -85,B 0,C 180,E1 13725.377,E2 13725.377} C_VEL
LIN {X 0,Y 473.911,Z 1002.085,A -85,B 0,C 180,E1 13723.642,E2 13723.642} C_VEL
LIN {X 0,Y 479.533,Z 983.861,A -85,B 0,C 180,E1 13722.251,E2 13722.251} C_VEL
LIN {X 0,Y 485.421,Z 963.289,A -85,B 0,C 180,E1 13720.892,E2 13720.892} C_VEL
LIN {X 0,Y 491.538,Z 939.198,A -85,B 0,C 180,E1 13719.561,E2 13719.561} C_VEL
LIN {X 0,Y 496,Z 919.238,A -85,B 0,C 180,E1 13718.634,E2 13718.634} C_VEL
LIN {X 0,Y 500.036,Z 898.674,A -85,B 0,C 180,E1 13717.829,E2 13717.829} C_VEL
LIN {X 0,Y 504.356,Z 872.769,A -85,B 0,C 180,E1 13717.013,E2 13717.013} C_VEL
LIN {X 0,Y 507.501,Z 847.712,A -85,B 0,C 180,E1 13716.425,E2 13716.425} C_VEL
LIN {X 0,Y 509.467,Z 825.598,A -85,B 0,C 180,E1 13716.024,E2 13716.024} C_VEL
LIN {X 0,Y 522.278,Z 592.966,A -85,B 0,C 180,E1 13712.499,E2 13712.499} C_VEL
LIN {X 0,Y 527.73,Z 498.444,A -85,B 0,C 180,E1 13711.054,E2 13711.054} C_VEL
LIN {X 0,Y 518.783,Z 483.582,A -85,B 0,C 180,E1 13708.775,E2 13708.775} C_VEL
LIN {X 0,Y 511.273,Z 471.749,A -85,B 0,C 180,E1 13706.663,E2 13706.663} C_VEL
LIN {X 0,Y 503.722,Z 460.287,A -85,B 0,C 180,E1 13704.292,E2 13704.292} C_VEL
LIN {X 0,Y 497.548,Z 451.252,A -85,B 0,C 180,E1 13702.109,E2 13702.109} C_VEL
LIN {X 0,Y 493.64,Z 445.759,A -85,B 0,C 180,E1 13700.575,E2 13700.575} C_VEL
LIN {X 0,Y 489.732,Z 440.234,A -85,B 0,C 180,E1 13698.882,E2 13698.882} C_VEL
LIN {X 0,Y 485.848,Z 435.003,A -85,B 0,C 180,E1 13696.992,E2 13696.992} C_VEL
LIN {X 0,Y 483.642,Z 431.75,A -85,B 0,C 180,E1 13695.775,E2 13695.775} C_VEL
LIN {X 0,Y 479.672,Z 426.428,A -85,B 0,C 180,E1 13693.256,E2 13693.256} C_VEL
LIN {X 0,Y 476.083,Z 421.404,A -85,B 0,C 180,E1 13690.284,E2 13690.284} C_VEL
LIN {X 0,Y 472.61,Z 416.273,A -85,B 0,C 180,E1 13685.22,E2 13685.22} C_VEL
LIN {X 0,Y 472.151,Z 415.527,A -85,B 0,C 180,E1 13680.728,E2 13680.728} C_VEL
LIN {X 0,Y 474.447,Z 416.98,A -85,B 0,C 180,E1 13676.133,E2 13676.133} C_VEL
LIN {X 0,Y 480.18,Z 423.421,A -85,B 0,C 180,E1 13670.955,E2 13670.955} C_VEL
LIN {X 0,Y 484.45,Z 428.367,A -85,B 0,C 180,E1 13668.33,E2 13668.33} C_VEL
LIN {X 0,Y 489.074,Z 433.988,A -85,B 0,C 180,E1 13665.979,E2 13665.979} C_VEL
LIN {X 0,Y 494.51,Z 440.88,A -85,B 0,C 180,E1 13663.616,E2 13663.616} C_VEL
LIN {X 0,Y 499.199,Z 446.94,A -85,B 0,C 180,E1 13661.822,E2 13661.822} C_VEL
LIN {X 0,Y 503.478,Z 452.577,A -85,B 0,C 180,E1 13660.329,E2 13660.329} C_VEL
LIN {X 0,Y 510.199,Z 461.62,A -85,B 0,C 180,E1 13658.199,E2 13658.199} C_VEL
LIN {X 0,Y 519.175,Z 474.35,A -85,B 0,C 180,E1 13655.66,E2 13655.66} C_VEL
LIN {X 0,Y 527.949,Z 487.823,A -85,B 0,C 180,E1 13653.42,E2 13653.42} C_VEL
LIN {X 0,Y 530.904,Z 492.757,A -85,B 0,C 180,E1 13652.706,E2 13652.706} C_VEL
LIN {X 0,Y 517.996,Z 705.703,A -85,B 0,C 180,E1 13649.339,E2 13649.339} C_VEL
LIN {X 0,Y 510.741,Z 827.023,A -85,B 0,C 180,E1 13647.403,E2 13647.403} C_VEL
LIN {X 0,Y 507.905,Z 854.599,A -85,B 0,C 180,E1 13646.854,E2 13646.854} C_VEL
LIN {X 0,Y 504.189,Z 880.209,A -85,B 0,C 180,E1 13646.162,E2 13646.162} C_VEL
LIN {X 0,Y 500.592,Z 901.006,A -85,B 0,C 180,E1 13645.469,E2 13645.469} C_VEL
LIN {X 0,Y 496.516,Z 921.635,A -85,B 0,C 180,E1 13644.645,E2 13644.645} C_VEL
LIN {X 0,Y 491.464,Z 944.303,A -85,B 0,C 180,E1 13643.575,E2 13643.575} C_VEL
LIN {X 0,Y 484.803,Z 970.608,A -85,B 0,C 180,E1 13642.076,E2 13642.076} C_VEL
LIN {X 0,Y 479.432,Z 989.919,A -85,B 0,C 180,E1 13640.785,E2 13640.785} C_VEL
LIN {X 0,Y 474.028,Z 1008.057,A -85,B 0,C 180,E1 13639.407,E2 13639.407} C_VEL
LIN {X 0,Y 468.221,Z 1026.512,A -85,B 0,C 180,E1 13637.817,E2 13637.817} C_VEL
LIN {X 0,Y 460.963,Z 1048.676,A -85,B 0,C 180,E1 13635.62,E2 13635.62} C_VEL
LIN {X 0,Y 454.262,Z 1068.054,A -85,B 0,C 180,E1 13633.372,E2 13633.372} C_VEL
LIN {X 0,Y 448.861,Z 1083.477,A -85,B 0,C 180,E1 13631.348,E2 13631.348} C_VEL
LIN {X 0,Y 443.584,Z 1098.49,A -85,B 0,C 180,E1 13629.134,E2 13629.134} C_VEL
LIN {X 0,Y 437.552,Z 1115.892,A -85,B 0,C 180,E1 13626.227,E2 13626.227} C_VEL
LIN {X 0,Y 432.081,Z 1131.823,A -85,B 0,C 180,E1 13623.1,E2 13623.1} C_VEL
LIN {X 0,Y 428.25,Z 1143.728,A -85,B 0,C 180,E1 13620.441,E2 13620.441} C_VEL
LIN {X 0,Y 424.865,Z 1154.89,A -85,B 0,C 180,E1 13617.621,E2 13617.621} C_VEL
LIN {X 0,Y 421.569,Z 1167.109,A -85,B 0,C 180,E1 13614.054,E2 13614.054} C_VEL
LIN {X 0,Y 419.269,Z 1176.783,A -85,B 0,C 180,E1 13610.668,E2 13610.668} C_VEL
LIN {X 0,Y 417.876,Z 1183.862,A -85,B 0,C 180,E1 13607.761,E2 13607.761} C_VEL
LIN {X 0,Y 416.947,Z 1189.805,A -85,B 0,C 180,E1 13604.868,E2 13604.868} C_VEL
LIN {X 0,Y 416.357,Z 1194.766,A -85,B 0,C 180,E1 13601.919,E2 13601.919} C_VEL
LIN {X 0,Y 416.055,Z 1198.943,A -85,B 0,C 180,E1 13598.708,E2 13598.708} C_VEL
LIN {X 0,Y 415.942,Z 1202.065,A -85,B 0,C 180,E1 13595.103,E2 13595.103} C_VEL
LIN {X 0,Y 415.926,Z 1203.421,A -85,B 0,C 180,E1 13591.928,E2 13591.928} C_VEL
LIN {X 0,Y 415.925,Z 1203.588,A -85,B 0,C 180,E1 13589.035,E2 13589.035} C_VEL
LIN {X 0,Y 415.929,Z 1202.779,A -85,B 0,C 180,E1 13586.278,E2 13586.278} C_VEL
LIN {X 0,Y 415.967,Z 1201.014,A -85,B 0,C 180,E1 13583.513,E2 13583.513} C_VEL
LIN {X 0,Y 416.087,Z 1198.279,A -85,B 0,C 180,E1 13580.735,E2 13580.735} C_VEL
LIN {X 0,Y 416.38,Z 1194.551,A -85,B 0,C 180,E1 13577.941,E2 13577.941} C_VEL
LIN {X 0,Y 416.952,Z 1189.771,A -85,B 0,C 180,E1 13575.113,E2 13575.113} C_VEL
LIN {X 0,Y 417.903,Z 1183.699,A -85,B 0,C 180,E1 13572.166,E2 13572.166} C_VEL
LIN {X 0,Y 419.357,Z 1176.37,A -85,B 0,C 180,E1 13569.174,E2 13569.174} C_VEL
LIN {X 0,Y 421.927,Z 1165.698,A -85,B 0,C 180,E1 13565.498,E2 13565.498} C_VEL
LIN {X 0,Y 425.079,Z 1154.153,A -85,B 0,C 180,E1 13562.184,E2 13562.184} C_VEL
LIN {X 0,Y 428.439,Z 1143.13,A -85,B 0,C 180,E1 13559.418,E2 13559.418} C_VEL
LIN {X 0,Y 432.52,Z 1130.492,A -85,B 0,C 180,E1 13556.619,E2 13556.619} C_VEL
LIN {X 0,Y 438.712,Z 1112.402,A -85,B 0,C 180,E1 13553.172,E2 13553.172} C_VEL
LIN {X 0,Y 443.88,Z 1097.589,A -85,B 0,C 180,E1 13550.73,E2 13550.73} C_VEL
LIN {X 0,Y 449.197,Z 1082.465,A -85,B 0,C 180,E1 13548.515,E2 13548.515} C_VEL
LIN {X 0,Y 455.727,Z 1063.847,A -85,B 0,C 180,E1 13546.107,E2 13546.107} C_VEL
LIN {X 0,Y 462.741,Z 1043.111,A -85,B 0,C 180,E1 13543.805,E2 13543.805} C_VEL
LIN {X 0,Y 468.891,Z 1024.271,A -85,B 0,C 180,E1 13541.985,E2 13541.985} C_VEL
LIN {X 0,Y 474.707,Z 1005.677,A -85,B 0,C 180,E1 13540.406,E2 13540.406} C_VEL
LIN {X 0,Y 481.621,Z 982.26,A -85,B 0,C 180,E1 13538.675,E2 13538.675} C_VEL
LIN {X 0,Y 487.963,Z 958.253,A -85,B 0,C 180,E1 13537.192,E2 13537.192} C_VEL
LIN {X 0,Y 492.76,Z 938.41,A -85,B 0,C 180,E1 13536.138,E2 13536.138} C_VEL
LIN {X 0,Y 497.044,Z 918.84,A -85,B 0,C 180,E1 13535.241,E2 13535.241} C_VEL
LIN {X 0,Y 501.46,Z 896.147,A -85,B 0,C 180,E1 13534.362,E2 13534.362} C_VEL
LIN {X 0,Y 506.046,Z 867.57,A -85,B 0,C 180,E1 13533.481,E2 13533.481} C_VEL
LIN {X 0,Y 508.933,Z 844.835,A -85,B 0,C 180,E1 13532.942,E2 13532.942} C_VEL
LIN {X 0,Y 511.04,Z 822.21,A -85,B 0,C 180,E1 13532.519,E2 13532.519} C_VEL
LIN {X 0,Y 523.795,Z 607.605,A -85,B 0,C 180,E1 13529.114,E2 13529.114} C_VEL
LIN {X 0,Y 530.759,Z 492.282,A -85,B 0,C 180,E1 13527.275,E2 13527.275} C_VEL
LIN {X 0,Y 521.088,Z 477.325,A -85,B 0,C 180,E1 13524.879,E2 13524.879} C_VEL
LIN {X 0,Y 511.939,Z 464.074,A -85,B 0,C 180,E1 13522.357,E2 13522.357} C_VEL
LIN {X 0,Y 503.829,Z 453.096,A -85,B 0,C 180,E1 13519.838,E2 13519.838} C_VEL
LIN {X 0,Y 499.279,Z 447.104,A -85,B 0,C 180,E1 13518.265,E2 13518.265} C_VEL
LIN {X 0,Y 495.893,Z 442.769,A -85,B 0,C 180,E1 13517,E2 13517} C_VEL
LIN {X 0,Y 492.723,Z 438.658,A -85,B 0,C 180,E1 13515.719,E2 13515.719} C_VEL
LIN {X 0,Y 488.646,Z 433.615,A -85,B 0,C 180,E1 13513.912,E2 13513.912} C_VEL
LIN {X 0,Y 484.797,Z 428.771,A -85,B 0,C 180,E1 13511.963,E2 13511.963} C_VEL
LIN {X 0,Y 480.064,Z 423.283,A -85,B 0,C 180,E1 13509.108,E2 13509.108} C_VEL
LIN {X 0,Y 474.303,Z 416.846,A -85,B 0,C 180,E1 13503.989,E2 13503.989} C_VEL
LIN {X 0,Y 471.88,Z 415.302,A -85,B 0,C 180,E1 13499.272,E2 13499.272} C_VEL
LIN {X 0,Y 472.299,Z 416.03,A -85,B 0,C 180,E1 13494.777,E2 13494.777} C_VEL
LIN {X 0,Y 473.005,Z 417.284,A -85,B 0,C 180,E1 13493.201,E2 13493.201} C_VEL
LIN {X 0,Y 476.732,Z 422.346,A -85,B 0,C 180,E1 13488.813,E2 13488.813} C_VEL
LIN {X 0,Y 480.629,Z 427.811,A -85,B 0,C 180,E1 13485.851,E2 13485.851} C_VEL
LIN {X 0,Y 484.548,Z 433.063,A -85,B 0,C 180,E1 13483.516,E2 13483.516} C_VEL
LIN {X 0,Y 491.237,Z 442.242,A -85,B 0,C 180,E1 13480.283,E2 13480.283} C_VEL
LIN {X 0,Y 496.803,Z 450.309,A -85,B 0,C 180,E1 13478.016,E2 13478.016} C_VEL
LIN {X 0,Y 502.461,Z 458.564,A -85,B 0,C 180,E1 13475.986,E2 13475.986} C_VEL
LIN {X 0,Y 507.514,Z 466.057,A -85,B 0,C 180,E1 13474.345,E2 13474.345} C_VEL
LIN {X 0,Y 515.378,Z 478.203,A -85,B 0,C 180,E1 13472.029,E2 13472.029} C_VEL
LIN {X 0,Y 524.697,Z 493.327,A -85,B 0,C 180,E1 13469.574,E2 13469.574} C_VEL
LIN {X 0,Y 527.674,Z 498.78,A -85,B 0,C 180,E1 13468.832,E2 13468.832} C_VEL
LIN {X 0,Y 514.606,Z 729.742,A -85,B 0,C 180,E1 13465.336,E2 13465.336} C_VEL
LIN {X 0,Y 508.975,Z 831.343,A -85,B 0,C 180,E1 13463.784,E2 13463.784} C_VEL
LIN {X 0,Y 506.139,Z 859.083,A -85,B 0,C 180,E1 13463.23,E2 13463.23} C_VEL
LIN {X 0,Y 502.947,Z 881.225,A -85,B 0,C 180,E1 13462.641,E2 13462.641} C_VEL
LIN {X 0,Y 499.327,Z 902.108,A -85,B 0,C 180,E1 13461.949,E2 13461.949} C_VEL
LIN {X 0,Y 494.391,Z 926.657,A -85,B 0,C 180,E1 13460.952,E2 13460.952} C_VEL
LIN {X 0,Y 488.651,Z 950.502,A -85,B 0,C 180,E1 13459.75,E2 13459.75} C_VEL
LIN {X 0,Y 483.36,Z 970.319,A -85,B 0,C 180,E1 13458.57,E2 13458.57} C_VEL
LIN {X 0,Y 477.053,Z 992.017,A -85,B 0,C 180,E1 13457.063,E2 13457.063} C_VEL
LIN {X 0,Y 470.058,Z 1013.677,A -85,B 0,C 180,E1 13455.273,E2 13455.273} C_VEL
LIN {X 0,Y 464.053,Z 1031.247,A -85,B 0,C 180,E1 13453.59,E2 13453.59} C_VEL
LIN {X 0,Y 457.461,Z 1049.751,A -85,B 0,C 180,E1 13451.557,E2 13451.557} C_VEL
LIN {X 0,Y 450.315,Z 1068.812,A -85,B 0,C 180,E1 13449.094,E2 13449.094} C_VEL
LIN {X 0,Y 444.696,Z 1083.551,A -85,B 0,C 180,E1 13446.894,E2 13446.894} C_VEL
LIN {X 0,Y 439.082,Z 1098.288,A -85,B 0,C 180,E1 13444.385,E2 13444.385} C_VEL
LIN {X 0,Y 433.196,Z 1113.801,A -85,B 0,C 180,E1 13441.288,E2 13441.288} C_VEL
LIN {X 0,Y 429.1,Z 1125.017,A -85,B 0,C 180,E1 13438.687,E2 13438.687} C_VEL
LIN {X 0,Y 425.329,Z 1135.944,A -85,B 0,C 180,E1 13435.779,E2 13435.779} C_VEL
LIN {X 0,Y 421.721,Z 1147.414,A -85,B 0,C 180,E1 13432.147,E2 13432.147} C_VEL
LIN {X 0,Y 419.576,Z 1155.176,A -85,B 0,C 180,E1 13429.2,E2 13429.2} C_VEL
LIN {X 0,Y 418.056,Z 1161.734,A -85,B 0,C 180,E1 13426.25,E2 13426.25} C_VEL
LIN {X 0,Y 417.04,Z 1167.11,A -85,B 0,C 180,E1 13423.326,E2 13423.326} C_VEL
LIN {X 0,Y 415.796,Z 1168.849,A -85,B 0,C 180,E1 13422.3,E2 13422.3} C_VEL
LIN {X 0,Y 408.949,Z 1172.897,A -85,B 0,C 180,E1 13419.471,E2 13419.471} C_VEL
LIN {X 0,Y 408.232,Z 1173.827,A -85,B 0,C 180,E1 13418.628,E2 13418.628} C_VEL
LIN {X 0,Y 407.999,Z 1176.816,A -85,B 0,C 180,E1 13414.921,E2 13414.921} C_VEL
LIN {X 0,Y 407.955,Z 1178.026,A -85,B 0,C 180,E1 13411.686,E2 13411.686} C_VEL
LIN {X 0,Y 407.96,Z 1178.126,A -85,B 0,C 180,E1 13408.877,E2 13408.877} C_VEL
LIN {X 0,Y 407.974,Z 1177.312,A -85,B 0,C 180,E1 13406.065,E2 13406.065} C_VEL
LIN {X 0,Y 408.078,Z 1175.575,A -85,B 0,C 180,E1 13403.246,E2 13403.246} C_VEL
LIN {X 0,Y 408.359,Z 1172.597,A -85,B 0,C 180,E1 13400.131,E2 13400.131} C_VEL
LIN {X 0,Y 409.142,Z 1167.323,A -85,B 0,C 180,E1 13396.288,E2 13396.288} C_VEL
LIN {X 0,Y 410.367,Z 1161.321,A -85,B 0,C 180,E1 13393,E2 13393} C_VEL
LIN {X 0,Y 412.066,Z 1154.654,A -85,B 0,C 180,E1 13389.993,E2 13389.993} C_VEL
LIN {X 0,Y 414.941,Z 1145.141,A -85,B 0,C 180,E1 13386.422,E2 13386.422} C_VEL
LIN {X 0,Y 418.507,Z 1134.554,A -85,B 0,C 180,E1 13383.157,E2 13383.157} C_VEL
LIN {X 0,Y 422.424,Z 1123.844,A -85,B 0,C 180,E1 13380.309,E2 13380.309} C_VEL
LIN {X 0,Y 428.042,Z 1109.413,A -85,B 0,C 180,E1 13377.025,E2 13377.025} C_VEL
LIN {X 0,Y 433.594,Z 1095.322,A -85,B 0,C 180,E1 13374.309,E2 13374.309} C_VEL
LIN {X 0,Y 439.078,Z 1081.581,A -85,B 0,C 180,E1 13371.993,E2 13371.993} C_VEL
LIN {X 0,Y 446.187,Z 1063.734,A -85,B 0,C 180,E1 13369.384,E2 13369.384} C_VEL
LIN {X 0,Y 452.982,Z 1045.882,A -85,B 0,C 180,E1 13367.168,E2 13367.168} C_VEL
LIN {X 0,Y 458.845,Z 1029.963,A -85,B 0,C 180,E1 13365.439,E2 13365.439} C_VEL
LIN {X 0,Y 465.557,Z 1010.932,A -85,B 0,C 180,E1 13363.633,E2 13363.633} C_VEL
LIN {X 0,Y 472.912,Z 988.309,A -85,B 0,C 180,E1 13361.816,E2 13361.816} C_VEL
LIN {X 0,Y 478.468,Z 969.673,A -85,B 0,C 180,E1 13360.536,E2 13360.536} C_VEL
LIN {X 0,Y 483.796,Z 950.216,A -85,B 0,C 180,E1 13359.38,E2 13359.38} C_VEL
LIN {X 0,Y 489.693,Z 926.27,A -85,B 0,C 180,E1 13358.177,E2 13358.177} C_VEL
LIN {X 0,Y 494.631,Z 902.381,A -85,B 0,C 180,E1 13357.208,E2 13357.208} C_VEL
LIN {X 0,Y 498.455,Z 880.886,A -85,B 0,C 180,E1 13356.498,E2 13356.498} C_VEL
LIN {X 0,Y 501.997,Z 856.788,A -85,B 0,C 180,E1 13355.864,E2 13355.864} C_VEL
LIN {X 0,Y 504.67,Z 830.228,A -85,B 0,C 180,E1 13355.348,E2 13355.348} C_VEL
LIN {X 0,Y 517.556,Z 605.023,A -85,B 0,C 180,E1 13351.918,E2 13351.918} C_VEL
LIN {X 0,Y 523.574,Z 502.761,A -85,B 0,C 180,E1 13350.34,E2 13350.34} C_VEL
LIN {X 0,Y 514.867,Z 488.117,A -85,B 0,C 180,E1 13348.033,E2 13348.033} C_VEL
LIN {X 0,Y 506.999,Z 475.634,A -85,B 0,C 180,E1 13345.714,E2 13345.714} C_VEL
LIN {X 0,Y 500.904,Z 466.419,A -85,B 0,C 180,E1 13343.718,E2 13343.718} C_VEL
LIN {X 0,Y 495.472,Z 458.318,A -85,B 0,C 180,E1 13341.735,E2 13341.735} C_VEL
LIN {X 0,Y 491.453,Z 452.589,A -85,B 0,C 180,E1 13340.111,E2 13340.111} C_VEL
LIN {X 0,Y 487.903,Z 447.46,A -85,B 0,C 180,E1 13338.521,E2 13338.521} C_VEL
LIN {X 0,Y 482.271,Z 439.453,A -85,B 0,C 180,E1 13335.575,E2 13335.575} C_VEL
LIN {X 0,Y 478.375,Z 434.143,A -85,B 0,C 180,E1 13333.046,E2 13333.046} C_VEL
LIN {X 0,Y 474.993,Z 429.287,A -85,B 0,C 180,E1 13330.185,E2 13330.185} C_VEL
LIN {X 0,Y 471.59,Z 424.176,A -85,B 0,C 180,E1 13325.109,E2 13325.109} C_VEL
LIN {X 0,Y 471.198,Z 423.473,A -85,B 0,C 180,E1 13320.608,E2 13320.608} C_VEL
LIN {X 0,Y 473.468,Z 424.943,A -85,B 0,C 180,E1 13316.125,E2 13316.125} C_VEL
LIN {X 0,Y 478.935,Z 431.235,A -85,B 0,C 180,E1 13311.113,E2 13311.113} C_VEL
LIN {X 0,Y 483.761,Z 437.028,A -85,B 0,C 180,E1 13308.132,E2 13308.132} C_VEL
LIN {X 0,Y 488.55,Z 443.009,A -85,B 0,C 180,E1 13305.722,E2 13305.722} C_VEL
LIN {X 0,Y 492.956,Z 448.614,A -85,B 0,C 180,E1 13303.805,E2 13303.805} C_VEL
LIN {X 0,Y 497.517,Z 454.589,A -85,B 0,C 180,E1 13302.031,E2 13302.031} C_VEL
LIN {X 0,Y 503.532,Z 462.521,A -85,B 0,C 180,E1 13299.938,E2 13299.938} C_VEL
LIN {X 0,Y 512.378,Z 474.999,A -85,B 0,C 180,E1 13297.209,E2 13297.209} C_VEL
LIN {X 0,Y 521.602,Z 488.808,A -85,B 0,C 180,E1 13294.692,E2 13294.692} C_VEL
LIN {X 0,Y 526.719,Z 497.193,A -85,B 0,C 180,E1 13293.398,E2 13293.398} C_VEL
LIN {X 0,Y 513.381,Z 711.18,A -85,B 0,C 180,E1 13290.006,E2 13290.006} C_VEL
LIN {X 0,Y 506.228,Z 827.09,A -85,B 0,C 180,E1 13288.15,E2 13288.15} C_VEL
LIN {X 0,Y 503.327,Z 854.654,A -85,B 0,C 180,E1 13287.601,E2 13287.601} C_VEL
LIN {X 0,Y 499.536,Z 880.142,A -85,B 0,C 180,E1 13286.914,E2 13286.914} C_VEL
LIN {X 0,Y 495.735,Z 901.544,A -85,B 0,C 180,E1 13286.2,E2 13286.2} C_VEL
LIN {X 0,Y 491.525,Z 922.226,A -85,B 0,C 180,E1 13285.37,E2 13285.37} C_VEL
LIN {X 0,Y 485.815,Z 947.102,A -85,B 0,C 180,E1 13284.184,E2 13284.184} C_VEL
LIN {X 0,Y 479.248,Z 971.865,A -85,B 0,C 180,E1 13282.744,E2 13282.744} C_VEL
LIN {X 0,Y 473.719,Z 991.084,A -85,B 0,C 180,E1 13281.445,E2 13281.445} C_VEL
LIN {X 0,Y 467.99,Z 1009.655,A -85,B 0,C 180,E1 13280.015,E2 13280.015} C_VEL
LIN {X 0,Y 460.677,Z 1032.193,A -85,B 0,C 180,E1 13278.02,E2 13278.02} C_VEL
LIN {X 0,Y 453.448,Z 1052.889,A -85,B 0,C 180,E1 13275.859,E2 13275.859} C_VEL
LIN {X 0,Y 447.594,Z 1069.235,A -85,B 0,C 180,E1 13273.917,E2 13273.917} C_VEL
LIN {X 0,Y 442.001,Z 1084.605,A -85,B 0,C 180,E1 13271.861,E2 13271.861} C_VEL
LIN {X 0,Y 435.81,Z 1101.613,A -85,B 0,C 180,E1 13269.288,E2 13269.288} C_VEL
LIN {X 0,Y 429.474,Z 1118.904,A -85,B 0,C 180,E1 13266.252,E2 13266.252} C_VEL
LIN {X 0,Y 424.73,Z 1132.29,A -85,B 0,C 180,E1 13263.552,E2 13263.552} C_VEL
LIN {X 0,Y 420.794,Z 1143.998,A -85,B 0,C 180,E1 13260.88,E2 13260.88} C_VEL
LIN {X 0,Y 416.952,Z 1156.174,A -85,B 0,C 180,E1 13257.724,E2 13257.724} C_VEL
LIN {X 0,Y 413.484,Z 1168.43,A -85,B 0,C 180,E1 13253.969,E2 13253.969} C_VEL
LIN {X 0,Y 411.409,Z 1176.851,A -85,B 0,C 180,E1 13250.932,E2 13250.932} C_VEL
LIN {X 0,Y 409.951,Z 1183.888,A -85,B 0,C 180,E1 13247.967,E2 13247.967} C_VEL
LIN {X 0,Y 408.946,Z 1190.046,A -85,B 0,C 180,E1 13244.876,E2 13244.876} C_VEL
LIN {X 0,Y 408.286,Z 1195.56,A -85,B 0,C 180,E1 13241.441,E2 13241.441} C_VEL
LIN {X 0,Y 408.008,Z 1199.798,A -85,B 0,C 180,E1 13237.746,E2 13237.746} C_VEL
LIN {X 0,Y 407.938,Z 1202.098,A -85,B 0,C 180,E1 13234.639,E2 13234.639} C_VEL
LIN {X 0,Y 407.929,Z 1203.197,A -85,B 0,C 180,E1 13231.826,E2 13231.826} C_VEL
LIN {X 0,Y 407.929,Z 1203.34,A -85,B 0,C 180,E1 13229.017,E2 13229.017} C_VEL
LIN {X 0,Y 407.932,Z 1202.525,A -85,B 0,C 180,E1 13226.205,E2 13226.205} C_VEL
LIN {X 0,Y 407.97,Z 1200.75,A -85,B 0,C 180,E1 13223.385,E2 13223.385} C_VEL
LIN {X 0,Y 408.1,Z 1198.002,A -85,B 0,C 180,E1 13220.552,E2 13220.552} C_VEL
LIN {X 0,Y 408.426,Z 1194.171,A -85,B 0,C 180,E1 13217.639,E2 13217.639} C_VEL
LIN {X 0,Y 409.02,Z 1189.514,A -85,B 0,C 180,E1 13214.837,E2 13214.837} C_VEL
LIN {X 0,Y 410.036,Z 1183.403,A -85,B 0,C 180,E1 13211.812,E2 13211.812} C_VEL
LIN {X 0,Y 411.58,Z 1176.109,A -85,B 0,C 180,E1 13208.778,E2 13208.778} C_VEL
LIN {X 0,Y 414.312,Z 1165.383,A -85,B 0,C 180,E1 13205.018,E2 13205.018} C_VEL
LIN {X 0,Y 417.588,Z 1154.035,A -85,B 0,C 180,E1 13201.699,E2 13201.699} C_VEL
LIN {X 0,Y 420.986,Z 1143.397,A -85,B 0,C 180,E1 13198.976,E2 13198.976} C_VEL
LIN {X 0,Y 425.006,Z 1131.473,A -85,B 0,C 180,E1 13196.274,E2 13196.274} C_VEL
LIN {X 0,Y 430.579,Z 1115.989,A -85,B 0,C 180,E1 13193.193,E2 13193.193} C_VEL
LIN {X 0,Y 436.762,Z 1098.866,A -85,B 0,C 180,E1 13190.284,E2 13190.284} C_VEL
LIN {X 0,Y 442.337,Z 1083.611,A -85,B 0,C 180,E1 13188.003,E2 13188.003} C_VEL
LIN {X 0,Y 448.15,Z 1067.624,A -85,B 0,C 180,E1 13185.884,E2 13185.884} C_VEL
LIN {X 0,Y 455.516,Z 1047.05,A -85,B 0,C 180,E1 13183.492,E2 13183.492} C_VEL
LIN {X 0,Y 462.819,Z 1025.372,A -85,B 0,C 180,E1 13181.354,E2 13181.354} C_VEL
LIN {X 0,Y 468.827,Z 1006.815,A -85,B 0,C 180,E1 13179.759,E2 13179.759} C_VEL
LIN {X 0,Y 475.033,Z 986.515,A -85,B 0,C 180,E1 13178.231,E2 13178.231} C_VEL
LIN {X 0,Y 482.347,Z 960.246,A -85,B 0,C 180,E1 13176.557,E2 13176.557} C_VEL
LIN {X 0,Y 487.671,Z 938.909,A -85,B 0,C 180,E1 13175.412,E2 13175.412} C_VEL
LIN {X 0,Y 492.344,Z 918.116,A -85,B 0,C 180,E1 13174.459,E2 13174.459} C_VEL
LIN {X 0,Y 497.177,Z 893.832,A -85,B 0,C 180,E1 13173.529,E2 13173.529} C_VEL
LIN {X 0,Y 501.544,Z 866.707,A -85,B 0,C 180,E1 13172.709,E2 13172.709} C_VEL
LIN {X 0,Y 504.452,Z 844.219,A -85,B 0,C 180,E1 13172.182,E2 13172.182} C_VEL
LIN {X 0,Y 506.611,Z 821.262,A -85,B 0,C 180,E1 13171.755,E2 13171.755} C_VEL
LIN {X 0,Y 519.892,Z 604.206,A -85,B 0,C 180,E1 13168.303,E2 13168.303} C_VEL
LIN {X 0,Y 526.599,Z 496.823,A -85,B 0,C 180,E1 13166.592,E2 13166.592} C_VEL
LIN {X 0,Y 517.073,Z 481.991,A -85,B 0,C 180,E1 13164.141,E2 13164.141} C_VEL
LIN {X 0,Y 508.702,Z 469.886,A -85,B 0,C 180,E1 13161.747,E2 13161.747} C_VEL
LIN {X 0,Y 501.527,Z 460.015,A -85,B 0,C 180,E1 13159.448,E2 13159.448} C_VEL
LIN {X 0,Y 495.628,Z 451.983,A -85,B 0,C 180,E1 13157.312,E2 13157.312} C_VEL
LIN {X 0,Y 490.791,Z 445.903,A -85,B 0,C 180,E1 13155.358,E2 13155.358} C_VEL
LIN {X 0,Y 486.923,Z 441.062,A -85,B 0,C 180,E1 13153.599,E2 13153.599} C_VEL
LIN {X 0,Y 482.632,Z 435.737,A -85,B 0,C 180,E1 13151.351,E2 13151.351} C_VEL
LIN {X 0,Y 478.231,Z 430.442,A -85,B 0,C 180,E1 13148.537,E2 13148.537} C_VEL
LIN {X 0,Y 473.13,Z 424.667,A -85,B 0,C 180,E1 13143.756,E2 13143.756} C_VEL
LIN {X 0,Y 470.878,Z 423.239,A -85,B 0,C 180,E1 13139.148,E2 13139.148} C_VEL
LIN {X 0,Y 471.375,Z 424.025,A -85,B 0,C 180,E1 13134.645,E2 13134.645} C_VEL
LIN {X 0,Y 472.222,Z 425.755,A -85,B 0,C 180,E1 13132.823,E2 13132.823} C_VEL
LIN {X 0,Y 475.56,Z 430.163,A -85,B 0,C 180,E1 13128.969,E2 13128.969} C_VEL
LIN {X 0,Y 479.392,Z 435.665,A -85,B 0,C 180,E1 13125.998,E2 13125.998} C_VEL
LIN {X 0,Y 483.153,Z 440.797,A -85,B 0,C 180,E1 13123.715,E2 13123.715} C_VEL
LIN {X 0,Y 489.556,Z 449.728,A -85,B 0,C 180,E1 13120.554,E2 13120.554} C_VEL
LIN {X 0,Y 495.397,Z 458.296,A -85,B 0,C 180,E1 13118.137,E2 13118.137} C_VEL
LIN {X 0,Y 502.711,Z 469.036,A -85,B 0,C 180,E1 13115.53,E2 13115.53} C_VEL
LIN {X 0,Y 512.006,Z 483.567,A -85,B 0,C 180,E1 13112.65,E2 13112.65} C_VEL
LIN {X 0,Y 521.457,Z 499.206,A -85,B 0,C 180,E1 13110.077,E2 13110.077} C_VEL
LIN {X 0,Y 523.556,Z 503.157,A -85,B 0,C 180,E1 13109.534,E2 13109.534} C_VEL
LIN {X 0,Y 510.142,Z 732.962,A -85,B 0,C 180,E1 13106.046,E2 13106.046} C_VEL
LIN {X 0,Y 504.502,Z 831.312,A -85,B 0,C 180,E1 13104.538,E2 13104.538} C_VEL
LIN {X 0,Y 501.587,Z 859.104,A -85,B 0,C 180,E1 13103.982,E2 13103.982} C_VEL
LIN {X 0,Y 498.304,Z 881.291,A -85,B 0,C 180,E1 13103.394,E2 13103.394} C_VEL
LIN {X 0,Y 494.593,Z 902.161,A -85,B 0,C 180,E1 13102.703,E2 13102.703} C_VEL
LIN {X 0,Y 489.658,Z 926.071,A -85,B 0,C 180,E1 13101.734,E2 13101.734} C_VEL
LIN {X 0,Y 483.767,Z 950.057,A -85,B 0,C 180,E1 13100.532,E2 13100.532} C_VEL
LIN {X 0,Y 478.352,Z 969.845,A -85,B 0,C 180,E1 13099.356,E2 13099.356} C_VEL
LIN {X 0,Y 472.408,Z 989.754,A -85,B 0,C 180,E1 13097.98,E2 13097.98} C_VEL
LIN {X 0,Y 464.84,Z 1012.765,A -85,B 0,C 180,E1 13096.104,E2 13096.104} C_VEL
LIN {X 0,Y 458.619,Z 1030.434,A -85,B 0,C 180,E1 13094.415,E2 13094.415} C_VEL
LIN {X 0,Y 452.631,Z 1046.696,A -85,B 0,C 180,E1 13092.64,E2 13092.64} C_VEL
LIN {X 0,Y 445.298,Z 1065.858,A -85,B 0,C 180,E1 13090.23,E2 13090.23} C_VEL
LIN {X 0,Y 438.784,Z 1082.227,A -85,B 0,C 180,E1 13087.806,E2 13087.806} C_VEL
LIN {X 0,Y 433.159,Z 1096.354,A -85,B 0,C 180,E1 13085.408,E2 13085.408} C_VEL
LIN {X 0,Y 427.164,Z 1111.633,A -85,B 0,C 180,E1 13082.414,E2 13082.414} C_VEL
LIN {X 0,Y 422.068,Z 1124.754,A -85,B 0,C 180,E1 13079.366,E2 13079.366} C_VEL
LIN {X 0,Y 418.259,Z 1135.235,A -85,B 0,C 180,E1 13076.554,E2 13076.554} C_VEL
LIN {X 0,Y 414.493,Z 1146.519,A -85,B 0,C 180,E1 13073.004,E2 13073.004} C_VEL
LIN {X 0,Y 411.935,Z 1155.107,A -85,B 0,C 180,E1 13069.718,E2 13069.718} C_VEL
LIN {X 0,Y 410.277,Z 1161.722,A -85,B 0,C 180,E1 13066.707,E2 13066.707} C_VEL
LIN {X 0,Y 409.013,Z 1168.135,A -85,B 0,C 180,E1 13063.141,E2 13063.141} C_VEL
LIN {X 0,Y 408.335,Z 1172.798,A -85,B 0,C 180,E1 13059.585,E2 13059.585} C_VEL
LIN {X 0,Y 408.232,Z 1173.827,A -85,B 0,C 180,E1 13058.628,E2 13058.628} C_VEL
LIN {X 0,Y 407.164,Z 1174.934,A -85,B 0,C 180,E1 13057.559,E2 13057.559} C_VEL
LIN {X 0,Y 400.644,Z 1177.241,A -85,B 0,C 180,E1 13054.615,E2 13054.615} C_VEL
LIN {X 0,Y 399.979,Z 1177.638,A -85,B 0,C 180,E1 13053.743,E2 13053.743} C_VEL
LIN {X 0,Y 399.954,Z 1178.424,A -85,B 0,C 180,E1 13050.717,E2 13050.717} C_VEL
LIN {X 0,Y 399.972,Z 1178.079,A -85,B 0,C 180,E1 13047.134,E2 13047.134} C_VEL
LIN {X 0,Y 400.058,Z 1176.258,A -85,B 0,C 180,E1 13043.687,E2 13043.687} C_VEL
LIN {X 0,Y 400.304,Z 1173.579,A -85,B 0,C 180,E1 13040.626,E2 13040.626} C_VEL
LIN {X 0,Y 400.808,Z 1169.918,A -85,B 0,C 180,E1 13037.612,E2 13037.612} C_VEL
LIN {X 0,Y 401.901,Z 1164.416,A -85,B 0,C 180,E1 13034.118,E2 13034.118} C_VEL
LIN {X 0,Y 403.768,Z 1156.958,A -85,B 0,C 180,E1 13030.47,E2 13030.47} C_VEL
LIN {X 0,Y 406.048,Z 1149.385,A -85,B 0,C 180,E1 13027.41,E2 13027.41} C_VEL
LIN {X 0,Y 409.064,Z 1140.542,A -85,B 0,C 180,E1 13024.365,E2 13024.365} C_VEL
LIN {X 0,Y 413.915,Z 1127.611,A -85,B 0,C 180,E1 13020.635,E2 13020.635} C_VEL
LIN {X 0,Y 418.515,Z 1116.011,A -85,B 0,C 180,E1 13017.808,E2 13017.808} C_VEL
LIN {X 0,Y 423.633,Z 1103.58,A -85,B 0,C 180,E1 13015.168,E2 13015.168} C_VEL
LIN {X 0,Y 430.795,Z 1086.352,A -85,B 0,C 180,E1 13012.044,E2 13012.044} C_VEL
LIN {X 0,Y 436.758,Z 1071.836,A -85,B 0,C 180,E1 13009.791,E2 13009.791} C_VEL
LIN {X 0,Y 443.058,Z 1056.254,A -85,B 0,C 180,E1 13007.672,E2 13007.672} C_VEL
LIN {X 0,Y 450.861,Z 1036.302,A -85,B 0,C 180,E1 13005.331,E2 13005.331} C_VEL
LIN {X 0,Y 457.85,Z 1017.23,A -85,B 0,C 180,E1 13003.437,E2 13003.437} C_VEL
LIN {X 0,Y 463.932,Z 999.699,A -85,B 0,C 180,E1 13001.923,E2 13001.923} C_VEL
LIN {X 0,Y 471.114,Z 977.558,A -85,B 0,C 180,E1 13000.272,E2 13000.272} C_VEL
LIN {X 0,Y 477.664,Z 954.718,A -85,B 0,C 180,E1 12998.859,E2 12998.859} C_VEL
LIN {X 0,Y 482.933,Z 934.431,A -85,B 0,C 180,E1 12997.796,E2 12997.796} C_VEL
LIN {X 0,Y 487.614,Z 914.202,A -85,B 0,C 180,E1 12996.898,E2 12996.898} C_VEL
LIN {X 0,Y 492.703,Z 888.26,A -85,B 0,C 180,E1 12995.957,E2 12995.957} C_VEL
LIN {X 0,Y 496.16,Z 866.456,A -85,B 0,C 180,E1 12995.334,E2 12995.334} C_VEL
LIN {X 0,Y 498.885,Z 844.907,A -85,B 0,C 180,E1 12994.849,E2 12994.849} C_VEL
LIN {X 0,Y 501.158,Z 818.65,A -85,B 0,C 180,E1 12994.388,E2 12994.388} C_VEL
LIN {X 0,Y 514.692,Z 586.924,A -85,B 0,C 180,E1 12990.863,E2 12990.863} C_VEL
LIN {X 0,Y 519.602,Z 507.238,A -85,B 0,C 180,E1 12989.641,E2 12989.641} C_VEL
LIN {X 0,Y 511.294,Z 493.267,A -85,B 0,C 180,E1 12987.359,E2 12987.359} C_VEL
LIN {X 0,Y 504.232,Z 481.914,A -85,B 0,C 180,E1 12985.205,E2 12985.205} C_VEL
LIN {X 0,Y 498.675,Z 473.341,A -85,B 0,C 180,E1 12983.329,E2 12983.329} C_VEL
LIN {X 0,Y 493.147,Z 464.984,A -85,B 0,C 180,E1 12981.25,E2 12981.25} C_VEL
LIN {X 0,Y 487.431,Z 456.49,A -85,B 0,C 180,E1 12978.788,E2 12978.788} C_VEL
LIN {X 0,Y 481.111,Z 447.37,A -85,B 0,C 180,E1 12975.49,E2 12975.49} C_VEL
LIN {X 0,Y 477.081,Z 441.856,A -85,B 0,C 180,E1 12972.836,E2 12972.836} C_VEL
LIN {X 0,Y 473.905,Z 437.17,A -85,B 0,C 180,E1 12970.086,E2 12970.086} C_VEL
LIN {X 0,Y 470.618,Z 432.129,A -85,B 0,C 180,E1 12965.12,E2 12965.12} C_VEL
LIN {X 0,Y 470.222,Z 431.413,A -85,B 0,C 180,E1 12960.609,E2 12960.609} C_VEL
LIN {X 0,Y 472.486,Z 432.929,A -85,B 0,C 180,E1 12956.117,E2 12956.117} C_VEL
LIN {X 0,Y 477.694,Z 439.047,A -85,B 0,C 180,E1 12951.271,E2 12951.271} C_VEL
LIN {X 0,Y 482.346,Z 444.722,A -85,B 0,C 180,E1 12948.339,E2 12948.339} C_VEL
LIN {X 0,Y 487.059,Z 450.716,A -85,B 0,C 180,E1 12945.92,E2 12945.92} C_VEL
LIN {X 0,Y 491.275,Z 456.152,A -85,B 0,C 180,E1 12944.052,E2 12944.052} C_VEL
LIN {X 0,Y 496.062,Z 462.526,A -85,B 0,C 180,E1 12942.159,E2 12942.159} C_VEL
LIN {X 0,Y 501.936,Z 470.509,A -85,B 0,C 180,E1 12940.084,E2 12940.084} C_VEL
LIN {X 0,Y 509.996,Z 481.995,A -85,B 0,C 180,E1 12937.553,E2 12937.553} C_VEL
LIN {X 0,Y 518.891,Z 495.511,A -85,B 0,C 180,E1 12935.069,E2 12935.069} C_VEL
LIN {X 0,Y 522.604,Z 501.782,A -85,B 0,C 180,E1 12934.097,E2 12934.097} C_VEL
LIN {X 0,Y 508.825,Z 716.694,A -85,B 0,C 180,E1 12930.685,E2 12930.685} C_VEL
LIN {X 0,Y 501.795,Z 827.269,A -85,B 0,C 180,E1 12928.909,E2 12928.909} C_VEL
LIN {X 0,Y 498.798,Z 854.965,A -85,B 0,C 180,E1 12928.355,E2 12928.355} C_VEL
LIN {X 0,Y 494.934,Z 880.306,A -85,B 0,C 180,E1 12927.674,E2 12927.674} C_VEL
LIN {X 0,Y 491.078,Z 901.494,A -85,B 0,C 180,E1 12926.967,E2 12926.967} C_VEL
LIN {X 0,Y 486.616,Z 922.824,A -85,B 0,C 180,E1 12926.111,E2 12926.111} C_VEL
LIN {X 0,Y 480.755,Z 947.585,A -85,B 0,C 180,E1 12924.925,E2 12924.925} C_VEL
LIN {X 0,Y 474.128,Z 971.86,A -85,B 0,C 180,E1 12923.508,E2 12923.508} C_VEL
LIN {X 0,Y 468.525,Z 990.758,A -85,B 0,C 180,E1 12922.23,E2 12922.23} C_VEL
LIN {X 0,Y 462.598,Z 1009.394,A -85,B 0,C 180,E1 12920.793,E2 12920.793} C_VEL
LIN {X 0,Y 455.144,Z 1031.657,A -85,B 0,C 180,E1 12918.818,E2 12918.818} C_VEL
LIN {X 0,Y 447.643,Z 1052.445,A -85,B 0,C 180,E1 12916.639,E2 12916.639} C_VEL
LIN {X 0,Y 441.548,Z 1068.857,A -85,B 0,C 180,E1 12914.679,E2 12914.679} C_VEL
LIN {X 0,Y 435.524,Z 1084.794,A -85,B 0,C 180,E1 12912.526,E2 12912.526} C_VEL
LIN {X 0,Y 428.438,Z 1103.555,A -85,B 0,C 180,E1 12909.632,E2 12909.632} C_VEL
LIN {X 0,Y 422.119,Z 1120.019,A -85,B 0,C 180,E1 12906.649,E2 12906.649} C_VEL
LIN {X 0,Y 417.411,Z 1132.76,A -85,B 0,C 180,E1 12904.021,E2 12904.021} C_VEL
LIN {X 0,Y 413.163,Z 1144.868,A -85,B 0,C 180,E1 12901.191,E2 12901.191} C_VEL
LIN {X 0,Y 408.726,Z 1158.411,A -85,B 0,C 180,E1 12897.539,E2 12897.539} C_VEL
LIN {X 0,Y 405.61,Z 1168.976,A -85,B 0,C 180,E1 12894.155,E2 12894.155} C_VEL
LIN {X 0,Y 403.559,Z 1176.928,A -85,B 0,C 180,E1 12891.207,E2 12891.207} C_VEL
LIN {X 0,Y 402.06,Z 1183.753,A -85,B 0,C 180,E1 12888.261,E2 12888.261} C_VEL
LIN {X 0,Y 401.021,Z 1189.768,A -85,B 0,C 180,E1 12885.177,E2 12885.177} C_VEL
LIN {X 0,Y 400.326,Z 1195.196,A -85,B 0,C 180,E1 12881.735,E2 12881.735} C_VEL
LIN {X 0,Y 400.017,Z 1199.539,A -85,B 0,C 180,E1 12877.902,E2 12877.902} C_VEL
LIN {X 0,Y 399.941,Z 1201.846,A -85,B 0,C 180,E1 12874.732,E2 12874.732} C_VEL
LIN {X 0,Y 399.933,Z 1202.949,A -85,B 0,C 180,E1 12871.862,E2 12871.862} C_VEL
LIN {X 0,Y 399.934,Z 1203.092,A -85,B 0,C 180,E1 12868.997,E2 12868.997} C_VEL
LIN {X 0,Y 399.935,Z 1202.274,A -85,B 0,C 180,E1 12866.129,E2 12866.129} C_VEL
LIN {X 0,Y 399.973,Z 1200.492,A -85,B 0,C 180,E1 12863.252,E2 12863.252} C_VEL
LIN {X 0,Y 400.116,Z 1197.737,A -85,B 0,C 180,E1 12860.361,E2 12860.361} C_VEL
LIN {X 0,Y 400.451,Z 1193.993,A -85,B 0,C 180,E1 12857.453,E2 12857.453} C_VEL
LIN {X 0,Y 401.102,Z 1189.235,A -85,B 0,C 180,E1 12854.53,E2 12854.53} C_VEL
LIN {X 0,Y 402.122,Z 1183.432,A -85,B 0,C 180,E1 12851.591,E2 12851.591} C_VEL
LIN {X 0,Y 403.647,Z 1176.552,A -85,B 0,C 180,E1 12848.645,E2 12848.645} C_VEL
LIN {X 0,Y 405.966,Z 1167.705,A -85,B 0,C 180,E1 12845.402,E2 12845.402} C_VEL
LIN {X 0,Y 409.853,Z 1154.79,A -85,B 0,C 180,E1 12841.434,E2 12841.434} C_VEL
LIN {X 0,Y 413.555,Z 1143.671,A -85,B 0,C 180,E1 12838.517,E2 12838.517} C_VEL
LIN {X 0,Y 417.75,Z 1131.803,A -85,B 0,C 180,E1 12835.773,E2 12835.773} C_VEL
LIN {X 0,Y 422.963,Z 1117.824,A -85,B 0,C 180,E1 12832.928,E2 12832.928} C_VEL
LIN {X 0,Y 429.915,Z 1099.483,A -85,B 0,C 180,E1 12829.717,E2 12829.717} C_VEL
LIN {X 0,Y 435.877,Z 1083.779,A -85,B 0,C 180,E1 12827.334,E2 12827.334} C_VEL
LIN {X 0,Y 441.897,Z 1067.843,A -85,B 0,C 180,E1 12825.197,E2 12825.197} C_VEL
LIN {X 0,Y 449.26,Z 1048.028,A -85,B 0,C 180,E1 12822.866,E2 12822.866} C_VEL
LIN {X 0,Y 456.768,Z 1026.592,A -85,B 0,C 180,E1 12820.718,E2 12820.718} C_VEL
LIN {X 0,Y 463.023,Z 1007.915,A -85,B 0,C 180,E1 12819.092,E2 12819.092} C_VEL
LIN {X 0,Y 469.065,Z 988.817,A -85,B 0,C 180,E1 12817.636,E2 12817.636} C_VEL
LIN {X 0,Y 475.881,Z 965.715,A -85,B 0,C 180,E1 12816.111,E2 12816.111} C_VEL
LIN {X 0,Y 482.193,Z 941.354,A -85,B 0,C 180,E1 12814.768,E2 12814.768} C_VEL
LIN {X 0,Y 486.995,Z 920.794,A -85,B 0,C 180,E1 12813.808,E2 12813.808} C_VEL
LIN {X 0,Y 491.36,Z 899.735,A -85,B 0,C 180,E1 12812.976,E2 12812.976} C_VEL
LIN {X 0,Y 495.651,Z 875.733,A -85,B 0,C 180,E1 12812.193,E2 12812.193} C_VEL
LIN {X 0,Y 499.6,Z 847.623,A -85,B 0,C 180,E1 12811.491,E2 12811.491} C_VEL
LIN {X 0,Y 501.932,Z 824.596,A -85,B 0,C 180,E1 12811.051,E2 12811.051} C_VEL
LIN {X 0,Y 515.178,Z 615.018,A -85,B 0,C 180,E1 12807.704,E2 12807.704} C_VEL
LIN {X 0,Y 522.478,Z 501.458,A -85,B 0,C 180,E1 12805.893,E2 12805.893} C_VEL
LIN {X 0,Y 513.784,Z 487.701,A -85,B 0,C 180,E1 12803.574,E2 12803.574} C_VEL
LIN {X 0,Y 504.778,Z 474.493,A -85,B 0,C 180,E1 12800.889,E2 12800.889} C_VEL
LIN {X 0,Y 496.813,Z 463.537,A -85,B 0,C 180,E1 12798.177,E2 12798.177} C_VEL
LIN {X 0,Y 492.198,Z 457.474,A -85,B 0,C 180,E1 12796.402,E2 12796.402} C_VEL
LIN {X 0,Y 489.01,Z 453.289,A -85,B 0,C 180,E1 12795.051,E2 12795.051} C_VEL
LIN {X 0,Y 485.457,Z 448.741,A -85,B 0,C 180,E1 12793.398,E2 12793.398} C_VEL
LIN {X 0,Y 481.231,Z 443.432,A -85,B 0,C 180,E1 12791.142,E2 12791.142} C_VEL
LIN {X 0,Y 476.913,Z 438.193,A -85,B 0,C 180,E1 12788.318,E2 12788.318} C_VEL
LIN {X 0,Y 472.152,Z 432.622,A -85,B 0,C 180,E1 12783.764,E2 12783.764} C_VEL
LIN {X 0,Y 469.903,Z 431.179,A -85,B 0,C 180,E1 12779.147,E2 12779.147} C_VEL
LIN {X 0,Y 470.403,Z 431.977,A -85,B 0,C 180,E1 12774.633,E2 12774.633} C_VEL
LIN {X 0,Y 471.969,Z 435.057,A -85,B 0,C 180,E1 12771.717,E2 12771.717} C_VEL
LIN {X 0,Y 474.393,Z 437.979,A -85,B 0,C 180,E1 12769.126,E2 12769.126} C_VEL
LIN {X 0,Y 478.076,Z 443.369,A -85,B 0,C 180,E1 12766.206,E2 12766.206} C_VEL
LIN {X 0,Y 481.764,Z 448.527,A -85,B 0,C 180,E1 12763.914,E2 12763.914} C_VEL
LIN {X 0,Y 487.887,Z 457.213,A -85,B 0,C 180,E1 12760.827,E2 12760.827} C_VEL
LIN {X 0,Y 494.212,Z 466.577,A -85,B 0,C 180,E1 12758.175,E2 12758.175} C_VEL
LIN {X 0,Y 502.05,Z 478.502,A -85,B 0,C 180,E1 12755.371,E2 12755.371} C_VEL
LIN {X 0,Y 510.463,Z 492.001,A -85,B 0,C 180,E1 12752.75,E2 12752.75} C_VEL
LIN {X 0,Y 519.221,Z 506.683,A -85,B 0,C 180,E1 12750.335,E2 12750.335} C_VEL
LIN {X 0,Y 519.514,Z 507.617,A -85,B 0,C 180,E1 12750.247,E2 12750.247} C_VEL
LIN {X 0,Y 505.729,Z 736.707,A -85,B 0,C 180,E1 12746.76,E2 12746.76} C_VEL
LIN {X 0,Y 500.105,Z 831.438,A -85,B 0,C 180,E1 12745.302,E2 12745.302} C_VEL
LIN {X 0,Y 497.062,Z 859.541,A -85,B 0,C 180,E1 12744.738,E2 12744.738} C_VEL
LIN {X 0,Y 493.726,Z 881.485,A -85,B 0,C 180,E1 12744.157,E2 12744.157} C_VEL
LIN {X 0,Y 489.89,Z 902.518,A -85,B 0,C 180,E1 12743.46,E2 12743.46} C_VEL
LIN {X 0,Y 484.751,Z 926.753,A -85,B 0,C 180,E1 12742.476,E2 12742.476} C_VEL
LIN {X 0,Y 478.704,Z 950.601,A -85,B 0,C 180,E1 12741.273,E2 12741.273} C_VEL
